C05463=1060.017,236.788,408.491,172.800,33.286,156.181
C05464=1060.024,237.036,408.463,172.802,33.289,156.182
C05465=1060.030,237.285,408.436,172.804,33.293,156.182
C05466=1060.036,237.533,408.408,172.807,33.297,156.183
C05467=1060.042,237.782,408.380,172.809,33.301,156.184
C05468=1060.048,238.030,408.353,172.811,33.305,156.185
C05469=1060.055,238.279,408.326,172.813,33.308,156.185
C05470=1060.061,238.527,408.298,172.815,33.312,156.186
C05471=1060.067,238.775,408.270,172.818,33.316,156.187
C05472=1060.073,239.024,408.243,172.820,33.320,156.188
C05473=1060.079,239.273,408.215,172.822,33.324,156.188
C05474=1060.085,239.521,408.187,172.824,33.328,156.189
C05475=1060.092,239.769,408.160,172.827,33.331,156.190
C05476=1060.098,240.017,408.132,172.829,33.335,156.190
C05477=1060.104,240.266,408.105,172.831,33.339,156.191
C05478=1060.110,240.515,408.077,172.833,33.343,156.192
C05479=1060.116,240.762,408.050,172.836,33.347,156.193
C05480=1060.122,241.011,408.021,172.838,33.350,156.193
C05481=1060.129,241.260,407.994,172.840,33.354,156.194
C05482=1060.135,241.507,407.966,172.842,33.358,156.195
C05483=1060.141,241.757,407.939,172.846,33.362,156.195
C05484=1060.147,242.005,407.911,172.848,33.365,156.196
C05485=1060.154,242.254,407.883,172.850,33.370,156.197
C05486=1060.159,242.502,407.855,172.852,33.373,156.198
C05487=1060.165,242.750,407.827,172.855,33.377,156.198
C05488=1060.171,242.998,407.800,172.857,33.381,156.199
C05489=1060.177,243.247,407.771,172.859,33.385,156.200
C05490=1060.184,243.495,407.743,172.861,33.389,156.201
C05491=1060.189,243.743,407.716,172.864,33.393,156.201
C05492=1060.196,243.992,407.688,172.866,33.396,156.202
C05493=1060.202,244.241,407.659,172.868,33.400,156.203
C05494=1060.209,244.489,407.632,172.870,33.404,156.204
C05495=1060.214,244.737,407.604,172.873,33.408,156.204
C05496=1060.221,244.986,407.576,172.875,33.412,156.205
C05497=1060.227,245.234,407.548,172.877,33.416,156.206
C05498=1060.232,245.482,407.520,172.880,33.420,156.206
C05499=1060.239,245.730,407.491,172.882,33.423,156.207
C05500=1060.245,245.979,407.463,172.885,33.427,156.208
C05501=1060.252,246.227,407.435,172.887,33.431,156.209
C05502=1060.257,246.475,407.407,172.890,33.435,156.209
C05503=1060.263,246.724,407.379,172.892,33.438,156.210
C05504=1060.270,246.973,407.351,172.894,33.443,156.211
C05505=1060.276,247.221,407.322,172.897,33.446,156.212
C05506=1060.281,247.469,407.294,172.899,33.451,156.212
C05507=1060.287,247.718,407.266,172.901,33.454,156.213
C05508=1060.293,247.966,407.238,172.904,33.458,156.214
C05509=1060.300,248.213,407.210,172.906,33.462,156.215
C05510=1060.305,248.462,407.181,172.908,33.466,156.215
C05511=1060.311,248.690,407.156,172.910,33.469,156.216
C05512=1060.316,248.917,407.130,172.912,33.473,156.217
C05513=1060.322,249.144,407.103,172.914,33.477,156.217
C05514=1060.327,249.372,407.078,172.917,33.480,156.218
C05515=1060.333,249.599,407.051,172.920,33.483,156.219
C05516=1060.338,249.825,407.025,172.922,33.487,156.219
C05517=1060.344,250.053,406.999,172.924,33.491,156.220
C05518=1060.350,250.281,406.974,172.926,33.494,156.221
C05519=1060.355,250.528,406.945,172.928,33.498,156.221
C05520=1060.361,250.777,406.917,172.931,33.502,156.222
C05521=1060.368,251.025,406.889,172.933,33.506,156.223
C05522=1060.374,251.273,406.860,172.935,33.509,156.224
C05523=1060.380,251.522,406.832,172.938,33.513,156.224
C05524=1060.386,251.770,406.803,172.940,33.517,156.225
C05525=1060.392,252.018,406.775,172.942,33.521,156.226
C05526=1060.398,252.267,406.745,172.945,33.525,156.227
C05527=1060.405,252.515,406.718,172.947,33.529,156.227
C05528=1060.411,252.763,406.689,172.950,33.532,156.228
C05529=1060.417,253.012,406.660,172.953,33.536,156.229
C05530=1060.423,253.260,406.631,172.955,33.540,156.230
C05531=1060.428,253.508,406.603,172.958,33.544,156.230
C05532=1060.435,253.756,406.574,172.960,33.548,156.231
C05533=1060.441,254.005,406.546,172.962,33.552,156.232
C05534=1060.448,254.253,406.518,172.965,33.555,156.232
C05535=1060.454,254.502,406.489,172.967,33.559,156.233
C05536=1060.460,254.750,406.460,172.970,33.563,156.234
C05537=1060.466,254.998,406.432,172.972,33.567,156.235
C05538=1060.472,255.247,406.403,172.974,33.571,156.235
C05539=1060.478,255.495,406.374,172.977,33.574,156.236
C05540=1060.484,255.743,406.345,172.979,33.578,156.237
C05541=1060.490,255.992,406.316,172.983,33.582,156.238
C05542=1060.497,256.239,406.288,172.985,33.586,156.238
C05543=1060.503,256.488,406.260,172.987,33.589,156.239
C05544=1060.510,256.736,406.231,172.990,33.594,156.240
C05545=1060.516,256.984,406.202,172.992,33.597,156.240
C05546=1060.522,257.233,406.173,172.995,33.601,156.241
C05547=1060.528,257.481,406.144,172.997,33.605,156.242
C05548=1060.534,257.729,406.115,172.999,33.609,156.243
C05549=1060.541,257.978,406.086,173.002,33.612,156.243
C05550=1060.547,258.226,406.058,173.004,33.616,156.244
C05551=1060.553,258.474,406.029,173.007,33.620,156.245
C05552=1060.560,258.722,406.000,173.009,33.624,156.246
C05553=1060.566,258.970,405.971,173.013,33.628,156.246
C05554=1060.572,259.218,405.942,173.015,33.631,156.247
C05555=1060.578,259.467,405.914,173.017,33.635,156.248
C05556=1060.584,259.715,405.885,173.020,33.639,156.249
C05557=1060.591,259.964,405.856,173.022,33.643,156.249
C05558=1060.597,260.212,405.827,173.025,33.646,156.250
C05559=1060.603,260.460,405.798,173.027,33.650,156.251
C05560=1060.609,260.708,405.769,173.030,33.654,156.251
C05561=1060.616,260.956,405.740,173.032,33.658,156.252
C05562=1060.622,261.204,405.711,173.035,33.662,156.253
C05563=1060.628,261.453,405.682,173.037,33.665,156.254
C05564=1060.635,261.702,405.653,173.041,33.669,156.254
C05565=1060.641,261.950,405.624,173.043,33.673,156.255
C05566=1060.647,262.198,405.595,173.045,33.677,156.256
C05567=1060.653,262.424,405.568,173.048,33.680,156.256
C05568=1060.659,262.650,405.542,173.050,33.683,156.257
C05569=1060.665,262.876,405.516,173.052,33.687,156.258
C05570=1060.671,263.103,405.489,173.055,33.690,156.258
C05571=1060.677,263.329,405.463,173.057,33.694,156.259
C05572=1060.682,263.555,405.436,173.059,33.697,156.260
C05573=1060.687,263.781,405.409,173.061,33.701,156.260
C05574=1060.693,264.007,405.382,173.064,33.704,156.261
C05575=1060.699,264.255,405.353,173.067,33.708,156.262
C05576=1060.705,264.503,405.324,173.069,33.712,156.263
C05577=1060.711,264.752,405.294,173.072,33.716,156.263
C05578=1060.717,264.999,405.265,173.074,33.720,156.264
C05579=1060.724,265.248,405.235,173.077,33.723,156.265
C05580=1060.731,265.496,405.206,173.079,33.727,156.266
C05581=1060.736,265.745,405.177,173.082,33.731,156.266
C05582=1060.742,265.993,405.148,173.084,33.735,156.267
C05583=1060.749,266.240,405.118,173.087,33.739,156.268
C05584=1060.754,266.489,405.088,173.089,33.743,156.268
C05585=1060.761,266.737,405.059,173.093,33.746,156.269
C05586=1060.767,266.986,405.030,173.095,33.750,156.270
C05587=1060.773,267.234,404.999,173.098,33.754,156.271
C05588=1060.780,267.482,404.970,173.100,33.758,156.271
C05589=1060.786,267.730,404.941,173.103,33.762,156.272
C05590=1060.792,267.978,404.911,173.106,33.766,156.273
C05591=1060.798,268.226,404.882,173.108,33.769,156.274
C05592=1060.805,268.475,404.852,173.111,33.773,156.274
C05593=1060.811,268.723,404.822,173.113,33.777,156.275
C05594=1060.817,268.971,404.793,173.117,33.781,156.276
C05595=1060.823,269.219,404.764,173.119,33.785,156.277
C05596=1060.829,269.467,404.734,173.122,33.788,156.277
C05597=1060.836,269.715,404.704,173.124,33.793,156.278
C05598=1060.842,269.963,404.674,173.127,33.796,156.279
C05599=1060.848,270.211,404.645,173.129,33.800,156.280
C05600=1060.854,270.459,404.615,173.132,33.804,156.280
C05601=1060.860,270.708,404.585,173.134,33.808,156.281
C05602=1060.866,270.956,404.555,173.137,33.811,156.282
C05603=1060.872,271.204,404.526,173.140,33.816,156.283
C05604=1060.878,271.452,404.495,173.143,33.819,156.283
C05605=1060.885,271.701,404.466,173.146,33.823,156.284
C05606=1060.891,271.948,404.436,173.148,33.827,156.285
C05607=1060.897,272.197,404.407,173.151,33.831,156.286
C05608=1060.903,272.444,404.376,173.153,33.835,156.286
C05609=1060.910,272.693,404.347,173.156,33.838,156.287
C05610=1060.916,272.941,404.316,173.158,33.843,156.288
C05611=1060.922,273.189,404.287,173.162,33.846,156.289
C05612=1060.928,273.438,404.257,173.165,33.850,156.289
C05613=1060.934,273.686,404.226,173.167,33.854,156.290
C05614=1060.941,273.933,404.197,173.170,33.858,156.291
C05615=1060.946,274.182,404.167,173.172,33.862,156.292
C05616=1060.953,274.430,404.137,173.175,33.866,156.292
C05617=1060.959,274.678,404.107,173.177,33.870,156.293
C05618=1060.965,274.925,404.076,173.180,33.873,156.294
C05619=1060.972,275.174,404.047,173.184,33.878,156.295
C05620=1060.978,275.422,404.016,173.186,33.881,156.295
C05621=1060.984,275.670,403.986,173.189,33.885,156.296
C05622=1060.991,275.918,403.956,173.191,33.889,156.297
C05623=1060.998,276.244,403.916,173.195,33.894,156.298
C05624=1061.006,276.568,403.877,173.198,33.899,156.299
C05625=1061.014,276.894,403.837,173.202,33.904,156.300
C05626=1061.023,277.219,403.798,173.206,33.909,156.301
C05627=1061.029,277.466,403.767,173.209,33.913,156.302
C05628=1061.035,277.715,403.737,173.211,33.917,156.303
C05629=1061.042,277.963,403.707,173.214,33.921,156.303
C05630=1061.047,278.210,403.677,173.217,33.925,156.304
C05631=1061.054,278.459,403.646,173.219,33.929,156.305
C05632=1061.059,278.707,403.616,173.222,33.932,156.305
C05633=1061.067,278.956,403.586,173.226,33.937,156.306
C05634=1061.072,279.203,403.556,173.228,33.940,156.307
C05635=1061.078,279.451,403.525,173.231,33.944,156.308
C05636=1061.085,279.700,403.495,173.233,33.948,156.309
C05637=1061.091,279.947,403.465,173.236,33.952,156.309
C05638=1061.098,280.196,403.434,173.239,33.956,156.310
C05639=1061.104,280.443,403.403,173.241,33.960,156.311
C05640=1061.110,280.691,403.372,173.244,33.964,156.312
C05641=1061.116,280.939,403.342,173.248,33.968,156.312
C05642=1061.122,281.188,403.311,173.250,33.972,156.313
C05643=1061.128,281.436,403.281,173.253,33.976,156.314
C05644=1061.134,281.683,403.251,173.256,33.980,156.315
C05645=1061.140,281.932,403.220,173.258,33.983,156.315
C05646=1061.146,282.180,403.190,173.261,33.987,156.316
C05647=1061.156,282.559,403.143,173.266,33.993,156.317
C05648=1061.166,282.938,403.095,173.270,33.999,156.319
C05649=1061.175,283.317,403.049,173.274,34.005,156.320
C05650=1061.185,283.696,403.002,173.278,34.011,156.321
C05651=1061.191,283.944,402.971,173.281,34.015,156.322
C05652=1061.197,284.192,402.940,173.285,34.019,156.323
C05653=1061.203,284.439,402.909,173.287,34.023,156.323
C05654=1061.210,284.688,402.879,173.290,34.027,156.324
C05655=1061.216,284.936,402.848,173.293,34.031,156.325
C05656=1061.222,285.184,402.817,173.296,34.035,156.326
C05657=1061.228,285.432,402.786,173.298,34.039,156.326
C05658=1061.235,285.679,402.755,173.301,34.043,156.327
C05659=1061.241,285.928,402.724,173.305,34.047,156.328
C05660=1061.247,286.176,402.694,173.307,34.051,156.329
C05661=1061.254,286.424,402.663,173.310,34.055,156.330
C05662=1061.260,286.672,402.632,173.313,34.059,156.330
C05663=1061.266,286.919,402.601,173.316,34.062,156.331
C05664=1061.273,287.168,402.570,173.318,34.067,156.332
C05665=1061.279,287.415,402.539,173.322,34.070,156.333
C05666=1061.285,287.664,402.508,173.325,34.074,156.333
C05667=1061.291,287.912,402.476,173.327,34.078,156.334
C05668=1061.297,288.160,402.446,173.330,34.082,156.335
C05669=1061.304,288.407,402.415,173.333,34.086,156.336
C05670=1061.310,288.656,402.384,173.336,34.090,156.337
C05671=1061.316,288.903,402.353,173.338,34.094,156.337
C05672=1061.323,289.152,402.322,173.342,34.098,156.338
C05673=1061.329,289.399,402.291,173.345,34.102,156.339
C05674=1061.335,289.647,402.259,173.348,34.106,156.340
C05675=1061.340,289.881,402.230,173.350,34.110,156.340
C05676=1061.347,290.114,402.201,173.353,34.114,156.341
C05677=1061.352,290.347,402.171,173.356,34.117,156.342
C05678=1061.358,290.581,402.142,173.359,34.121,156.343
C05679=1061.364,290.815,402.113,173.362,34.125,156.343
C05680=1061.370,291.048,402.083,173.364,34.129,156.344
C05681=1061.376,291.281,402.054,173.367,34.132,156.345
C05682=1061.382,291.515,402.023,173.370,34.136,156.346
C05683=1061.388,291.763,401.993,173.372,34.140,156.347
C05684=1061.394,292.011,401.962,173.376,34.144,156.347
C05685=1061.401,292.259,401.930,173.379,34.148,156.348
C05686=1061.407,292.507,401.898,173.382,34.152,156.349
C05687=1061.413,292.754,401.867,173.384,34.156,156.350
C05688=1061.420,293.002,401.836,173.387,34.160,156.351
C05689=1061.426,293.251,401.804,173.390,34.164,156.351
C05690=1061.432,293.498,401.773,173.394,34.168,156.352
C05691=1061.438,293.746,401.742,173.397,34.172,156.353
C05692=1061.444,293.994,401.710,173.399,34.176,156.354
C05693=1061.451,294.242,401.678,173.402,34.180,156.354
C05694=1061.457,294.489,401.647,173.405,34.184,156.355
C05695=1061.463,294.737,401.615,173.409,34.188,156.356
C05696=1061.470,294.985,401.584,173.412,34.192,156.357
C05697=1061.476,295.233,401.552,173.415,34.196,156.358
C05698=1061.483,295.481,401.520,173.417,34.200,156.359
C05699=1061.488,295.729,401.489,173.420,34.204,156.359
C05700=1061.495,295.977,401.457,173.423,34.209,156.360
C05701=1061.502,296.225,401.426,173.427,34.212,156.361
C05702=1061.508,296.473,401.394,173.430,34.216,156.362
C05703=1061.514,296.721,401.362,173.433,34.221,156.363
C05704=1061.520,296.968,401.331,173.435,34.225,156.363
C05705=1061.526,297.216,401.299,173.438,34.229,156.364
C05706=1061.532,297.464,401.267,173.442,34.233,156.365
C05707=1061.539,297.712,401.235,173.445,34.237,156.366
C05708=1061.544,297.959,401.203,173.448,34.241,156.367
C05709=1061.551,298.207,401.172,173.451,34.245,156.368
C05710=1061.557,298.456,401.139,173.453,34.250,156.368
C05711=1061.563,298.704,401.107,173.457,34.254,156.369
C05712=1061.568,298.951,401.075,173.460,34.258,156.370
C05713=1061.575,299.199,401.044,173.463,34.262,156.371
C05714=1061.581,299.447,401.012,173.466,34.266,156.372
C05715=1061.587,299.694,400.979,173.469,34.270,156.373
C05716=1061.593,299.943,400.947,173.471,34.274,156.373
C05717=1061.600,300.191,400.915,173.475,34.278,156.374
C05718=1061.606,300.437,400.883,173.478,34.282,156.375
C05719=1061.612,300.686,400.851,173.481,34.286,156.376
C05720=1061.618,300.934,400.819,173.484,34.291,156.377
C05721=1061.624,301.181,400.786,173.487,34.295,156.378
C05722=1061.631,301.429,400.755,173.491,34.299,156.378
C05723=1061.637,301.678,400.723,173.494,34.303,156.379
C05724=1061.643,301.925,400.690,173.497,34.307,156.380
C05725=1061.649,302.173,400.658,173.499,34.311,156.381
C05726=1061.656,302.420,400.626,173.503,34.315,156.382
C05727=1061.661,302.668,400.594,173.506,34.320,156.383
C05728=1061.668,302.916,400.561,173.509,34.324,156.383
C05729=1061.674,303.164,400.529,173.512,34.328,156.384
C05730=1061.680,303.412,400.497,173.515,34.332,156.385
C05731=1061.686,303.653,400.465,173.519,34.336,156.386
C05732=1061.693,303.894,400.434,173.522,34.340,156.387
C05733=1061.699,304.134,400.403,173.524,34.344,156.388
C05734=1061.704,304.376,400.371,173.527,34.349,156.388
C05735=1061.711,304.617,400.340,173.530,34.353,156.389
C05736=1061.718,304.858,400.308,173.534,34.357,156.390
C05737=1061.723,305.099,400.276,173.537,34.360,156.391
C05738=1061.729,305.340,400.245,173.540,34.365,156.392
C05739=1061.735,305.587,400.213,173.543,34.369,156.393
C05740=1061.741,305.836,400.181,173.546,34.373,156.393
C05741=1061.748,306.084,400.147,173.550,34.377,156.394
C05742=1061.755,306.331,400.115,173.553,34.381,156.395
C05743=1061.761,306.579,400.083,173.556,34.386,156.396
C05744=1061.768,306.827,400.051,173.559,34.390,156.397
C05745=1061.774,307.075,400.018,173.563,34.394,156.398
C05746=1061.780,307.322,399.985,173.566,34.398,156.399
C05747=1061.786,307.570,399.953,173.568,34.402,156.399
C05748=1061.793,307.818,399.920,173.571,34.407,156.400
C05749=1061.800,308.065,399.888,173.574,34.411,156.401
C05750=1061.806,308.313,399.855,173.578,34.415,156.402
C05751=1061.812,308.560,399.823,173.581,34.419,156.403
C05752=1061.818,308.808,399.790,173.584,34.423,156.404
C05753=1061.825,309.057,399.758,173.587,34.427,156.404
C05754=1061.831,309.305,399.725,173.591,34.431,156.405
C05755=1061.838,309.552,399.692,173.594,34.436,156.406
C05756=1061.844,309.800,399.659,173.597,34.440,156.407
C05757=1061.850,310.047,399.627,173.600,34.444,156.408
C05758=1061.858,310.295,399.594,173.603,34.448,156.409
C05759=1061.864,310.543,399.561,173.608,34.453,156.410
C05760=1061.870,310.790,399.529,173.611,34.457,156.410
C05761=1061.877,311.038,399.496,173.614,34.461,156.411
C05762=1061.883,311.286,399.463,173.617,34.465,156.412
C05763=1061.890,311.534,399.430,173.621,34.469,156.413
C05764=1061.896,311.782,399.397,173.624,34.474,156.414
C05765=1061.902,312.029,399.364,173.627,34.478,156.415
C05766=1061.909,312.277,399.332,173.630,34.482,156.416
C05767=1061.916,312.525,399.299,173.634,34.486,156.416
C05768=1061.922,312.773,399.266,173.637,34.490,156.417
C05769=1061.928,313.020,399.233,173.640,34.495,156.418
C05770=1061.935,313.268,399.199,173.643,34.499,156.419
C05771=1061.942,313.515,399.167,173.647,34.503,156.420
C05772=1061.948,313.763,399.134,173.650,34.507,156.421
C05773=1061.955,314.011,399.101,173.653,34.512,156.422
C05774=1061.961,314.259,399.068,173.656,34.516,156.423
C05775=1061.967,314.506,399.034,173.660,34.520,156.424
C05776=1061.973,314.754,399.001,173.663,34.525,156.424
C05777=1061.979,315.002,398.968,173.666,34.529,156.425
C05778=1061.986,315.249,398.934,173.669,34.534,156.426
C05779=1061.992,315.497,398.901,173.673,34.538,156.427
C05780=1061.998,315.745,398.868,173.676,34.543,156.428
C05781=1062.005,315.992,398.834,173.679,34.547,156.429
C05782=1062.011,316.240,398.801,173.683,34.552,156.430
C05783=1062.017,316.487,398.767,173.687,34.556,156.431
C05784=1062.023,316.735,398.734,173.690,34.560,156.432
C05785=1062.029,316.983,398.701,173.693,34.564,156.433
C05786=1062.036,317.231,398.667,173.696,34.569,156.434
C05787=1062.042,317.473,398.635,173.700,34.573,156.434
C05788=1062.048,317.716,398.601,173.703,34.578,156.435
C05789=1062.054,317.960,398.568,173.706,34.582,156.436
C05790=1062.060,318.202,398.535,173.709,34.586,156.437
C05791=1062.067,318.445,398.503,173.713,34.591,156.438
C05792=1062.073,318.688,398.470,173.716,34.595,156.439
C05793=1062.079,318.932,398.436,173.719,34.600,156.440
C05794=1062.085,319.174,398.404,173.722,34.604,156.441
C05795=1062.091,319.423,398.370,173.726,34.608,156.442
C05796=1062.097,319.670,398.336,173.729,34.612,156.443
C05797=1062.105,319.917,398.303,173.732,34.617,156.444
C05798=1062.110,320.165,398.269,173.736,34.621,156.444
C05799=1062.117,320.412,398.236,173.740,34.626,156.445
C05800=1062.123,320.660,398.201,173.743,34.631,156.446
C05801=1062.129,320.908,398.169,173.746,34.635,156.447
C05802=1062.136,321.156,398.134,173.750,34.639,156.448
C05803=1062.143,321.403,398.101,173.753,34.644,156.449
C05804=1062.149,321.651,398.066,173.756,34.648,156.450
C05805=1062.155,321.898,398.034,173.760,34.653,156.451
C05806=1062.162,322.146,397.999,173.764,34.657,156.452
C05807=1062.168,322.393,397.966,173.767,34.662,156.453
C05808=1062.175,322.641,397.931,173.770,34.666,156.454
C05809=1062.181,322.889,397.897,173.774,34.670,156.455
C05810=1062.188,323.137,397.864,173.777,34.675,156.456
C05811=1062.193,323.384,397.830,173.780,34.680,156.457
C05812=1062.201,323.632,397.796,173.785,34.684,156.457
C05813=1062.206,323.879,397.762,173.788,34.688,156.458
C05814=1062.214,324.127,397.728,173.791,34.693,156.459
C05815=1062.220,324.375,397.694,173.794,34.698,156.460
C05816=1062.226,324.622,397.660,173.798,34.702,156.461
C05817=1062.233,324.870,397.626,173.802,34.707,156.462
C05818=1062.239,325.117,397.592,173.805,34.711,156.463
C05819=1062.246,325.365,397.558,173.809,34.716,156.464
C05820=1062.253,325.613,397.524,173.812,34.720,156.465
C05821=1062.259,325.860,397.490,173.815,34.725,156.466
C05822=1062.266,326.108,397.456,173.820,34.729,156.467
C05823=1062.272,326.356,397.421,173.823,34.734,156.468
C05824=1062.279,326.603,397.388,173.826,34.738,156.469
C05825=1062.285,326.851,397.354,173.829,34.743,156.470
C05826=1062.292,327.099,397.319,173.833,34.747,156.471
C05827=1062.298,327.346,397.286,173.837,34.752,156.472
C05828=1062.305,327.593,397.251,173.840,34.756,156.473
C05829=1062.312,327.841,397.216,173.844,34.761,156.474
C05830=1062.318,328.088,397.183,173.847,34.765,156.475
C05831=1062.325,328.336,397.148,173.851,34.770,156.475
C05832=1062.331,328.584,397.114,173.855,34.775,156.476
C05833=1062.339,328.831,397.079,173.858,34.779,156.477
C05834=1062.344,329.078,397.045,173.861,34.783,156.478
C05835=1062.351,329.326,397.011,173.866,34.788,156.479
C05836=1062.358,329.574,396.977,173.869,34.793,156.480
C05837=1062.365,329.821,396.942,173.872,34.797,156.481
C05838=1062.371,330.069,396.907,173.876,34.802,156.482
C05839=1062.378,330.316,396.874,173.880,34.807,156.483
C05840=1062.385,330.564,396.839,173.883,34.811,156.484
C05841=1062.391,330.812,396.804,173.886,34.816,156.485
C05842=1062.398,331.060,396.770,173.891,34.821,156.486
C05843=1062.404,331.299,396.736,173.894,34.825,156.487
C05844=1062.411,331.540,396.703,173.897,34.830,156.488
C05845=1062.417,331.780,396.669,173.901,34.835,156.489
C05846=1062.423,332.020,396.635,173.904,34.839,156.490
C05847=1062.429,332.260,396.602,173.908,34.843,156.491
C05848=1062.436,332.500,396.568,173.912,34.848,156.492
C05849=1062.442,332.740,396.534,173.915,34.853,156.493
C05850=1062.448,332.980,396.501,173.918,34.857,156.494
C05851=1062.454,333.228,396.465,173.923,34.862,156.495
C05852=1062.461,333.474,396.430,173.926,34.867,156.496
C05853=1062.467,333.722,396.396,173.929,34.872,156.497
C05854=1062.474,333.970,396.361,173.934,34.876,156.498
C05855=1062.481,334.217,396.326,173.937,34.881,156.499
C05856=1062.487,334.465,396.291,173.940,34.886,156.500
C05857=1062.494,334.713,396.256,173.944,34.891,156.501
C05858=1062.501,334.960,396.221,173.948,34.895,156.502
C05859=1062.507,335.208,396.187,173.952,34.900,156.503
C05860=1062.513,335.455,396.152,173.956,34.905,156.504
C05861=1062.520,335.702,396.117,173.959,34.910,156.505
C05862=1062.527,335.949,396.082,173.963,34.914,156.506
C05863=1062.534,336.197,396.046,173.967,34.919,156.507
C05864=1062.540,336.445,396.012,173.970,34.924,156.508
C05865=1062.547,336.692,395.977,173.974,34.929,156.509
C05866=1062.553,336.940,395.941,173.978,34.934,156.510
C05867=1062.560,337.187,395.906,173.981,34.939,156.511
C05868=1062.566,337.434,395.871,173.985,34.943,156.512
C05869=1062.573,337.682,395.836,173.989,34.948,156.513
C05870=1062.579,337.929,395.800,173.992,34.953,156.514
C05871=1062.586,338.177,395.765,173.997,34.958,156.515
C05872=1062.593,338.424,395.730,174.000,34.963,156.516
C05873=1062.599,338.672,395.694,174.004,34.968,156.518
C05874=1062.605,338.919,395.659,174.008,34.973,156.519
C05875=1062.612,339.167,395.624,174.011,34.978,156.520
C05876=1062.618,339.414,395.588,174.016,34.983,156.521
C05877=1062.625,339.662,395.553,174.019,34.988,156.522
C05878=1062.632,339.909,395.518,174.023,34.993,156.523
C05879=1062.639,340.156,395.483,174.027,34.997,156.524
C05880=1062.645,340.403,395.446,174.030,35.003,156.525
C05881=1062.652,340.651,395.411,174.035,35.007,156.526
C05882=1062.658,340.898,395.376,174.038,35.012,156.527
C05883=1062.664,341.146,395.340,174.041,35.018,156.528
C05884=1062.671,341.393,395.305,174.046,35.022,156.529
C05885=1062.678,341.640,395.269,174.049,35.027,156.530
C05886=1062.684,341.888,395.233,174.054,35.033,156.531
C05887=1062.691,342.135,395.198,174.057,35.037,156.532
C05888=1062.698,342.383,395.162,174.061,35.042,156.534
C05889=1062.705,342.630,395.126,174.065,35.047,156.535
C05890=1062.712,342.877,395.091,174.069,35.052,156.536
C05891=1062.718,343.125,395.055,174.073,35.057,156.537
C05892=1062.725,343.372,395.020,174.077,35.062,156.538
C05893=1062.731,343.620,394.984,174.080,35.068,156.539
C05894=1062.738,343.867,394.948,174.085,35.072,156.540
C05895=1062.744,344.115,394.912,174.088,35.077,156.541
C05896=1062.751,344.361,394.876,174.092,35.083,156.542
C05897=1062.758,344.609,394.840,174.096,35.088,156.543
C05898=1062.765,344.856,394.805,174.100,35.093,156.545
C05899=1062.771,345.094,394.770,174.104,35.098,156.546
C05900=1062.778,345.332,394.735,174.107,35.103,156.547
C05901=1062.783,345.569,394.701,174.112,35.108,156.548
C05902=1062.790,345.807,394.666,174.115,35.112,156.549
C05903=1062.796,346.045,394.632,174.119,35.117,156.550
C05904=1062.802,346.282,394.597,174.123,35.123,156.551
C05905=1062.809,346.520,394.562,174.126,35.127,156.552
C05906=1062.815,346.758,394.528,174.130,35.132,156.553
C05907=1062.822,347.005,394.491,174.134,35.138,156.554
C05908=1062.829,347.252,394.455,174.138,35.143,156.555
C05909=1062.835,347.500,394.419,174.142,35.148,156.556
C05910=1062.842,347.748,394.383,174.147,35.153,156.558
C05911=1062.849,347.994,394.347,174.150,35.158,156.559
C05912=1062.855,348.241,394.310,174.154,35.163,156.560
C05913=1062.862,348.490,394.274,174.158,35.169,156.561
C05914=1062.869,348.736,394.239,174.162,35.174,156.562
C05915=1062.875,348.983,394.202,174.166,35.179,156.563
C05916=1062.882,349.231,394.165,174.170,35.184,156.564
C05917=1062.888,349.478,394.129,174.174,35.190,156.566
C05918=1062.895,349.725,394.093,174.178,35.195,156.567
C05919=1062.902,349.973,394.056,174.183,35.200,156.568
C05920=1062.909,350.220,394.020,174.186,35.205,156.569
C05921=1062.916,350.467,393.984,174.191,35.211,156.570
C05922=1062.923,350.714,393.947,174.194,35.216,156.571
C05923=1062.929,350.961,393.911,174.198,35.221,156.573
C05924=1062.936,351.209,393.874,174.203,35.227,156.574
C05925=1062.943,351.456,393.838,174.206,35.232,156.575
C05926=1062.950,351.704,393.801,174.211,35.237,156.576
C05927=1062.956,351.951,393.765,174.214,35.243,156.577
C05928=1062.963,352.198,393.728,174.219,35.248,156.578
C05929=1062.970,352.446,393.691,174.223,35.253,156.580
C05930=1062.976,352.693,393.655,174.227,35.258,156.581
C05931=1062.983,352.940,393.617,174.231,35.264,156.582
C05932=1062.990,353.187,393.581,174.235,35.269,156.583
C05933=1062.996,353.434,393.545,174.239,35.275,156.584
C05934=1063.003,353.682,393.508,174.244,35.280,156.586
C05935=1063.009,353.928,393.471,174.247,35.286,156.587
C05936=1063.016,354.176,393.434,174.252,35.291,156.588
C05937=1063.023,354.423,393.397,174.256,35.297,156.589
C05938=1063.030,354.670,393.360,174.260,35.302,156.590
C05939=1063.036,354.917,393.323,174.264,35.307,156.592
C05940=1063.043,355.165,393.287,174.269,35.313,156.593
C05941=1063.050,355.411,393.249,174.272,35.319,156.594
C05942=1063.057,355.659,393.213,174.277,35.324,156.595
C05943=1063.063,355.905,393.175,174.281,35.330,156.596
C05944=1063.070,356.153,393.139,174.285,35.335,156.598
C05945=1063.078,356.400,393.101,174.289,35.340,156.599
C05946=1063.084,356.647,393.065,174.294,35.346,156.600
C05947=1063.091,356.894,393.027,174.297,35.352,156.601
C05948=1063.098,357.142,392.991,174.302,35.357,156.603
C05949=1063.105,357.389,392.953,174.306,35.363,156.604
C05950=1063.112,357.636,392.916,174.311,35.368,156.605
C05951=1063.118,357.883,392.879,174.314,35.374,156.606
C05952=1063.126,358.130,392.842,174.319,35.379,156.608
C05953=1063.133,358.378,392.805,174.323,35.385,156.609
C05954=1063.139,358.624,392.768,174.327,35.391,156.610
C05955=1063.146,358.864,392.731,174.331,35.396,156.611
C05956=1063.152,359.104,392.695,174.336,35.401,156.612
C05957=1063.159,359.343,392.659,174.340,35.407,156.614
C05958=1063.166,359.584,392.622,174.344,35.413,156.615
C05959=1063.173,359.823,392.586,174.349,35.418,156.616
C05960=1063.179,360.063,392.550,174.352,35.423,156.617
C05961=1063.186,360.303,392.513,174.357,35.429,156.619
C05962=1063.193,360.543,392.478,174.361,35.435,156.620
C05963=1063.199,360.790,392.439,174.365,35.440,156.621
C05964=1063.206,361.037,392.402,174.369,35.446,156.622
C05965=1063.213,361.284,392.365,174.374,35.452,156.624
C05966=1063.220,361.531,392.327,174.378,35.457,156.625
C05967=1063.227,361.778,392.289,174.382,35.463,156.626
C05968=1063.233,362.025,392.252,174.387,35.469,156.628
C05969=1063.241,362.272,392.214,174.391,35.475,156.629
C05970=1063.247,362.520,392.176,174.396,35.480,156.630
C05971=1063.254,362.767,392.139,174.400,35.486,156.631
C05972=1063.261,363.013,392.102,174.404,35.492,156.633
C05973=1063.268,363.260,392.064,174.408,35.498,156.634
C05974=1063.275,363.508,392.026,174.413,35.504,156.635
C05975=1063.282,363.754,391.988,174.418,35.509,156.637
C05976=1063.290,364.001,391.950,174.422,35.515,156.638
C05977=1063.296,364.249,391.912,174.426,35.521,156.639
C05978=1063.303,364.495,391.875,174.430,35.527,156.641
C05979=1063.309,364.743,391.837,174.435,35.533,156.642
C05980=1063.317,364.989,391.798,174.440,35.539,156.643
C05981=1063.323,365.237,391.760,174.444,35.545,156.645
C05982=1063.330,365.484,391.722,174.449,35.551,156.646
C05983=1063.337,365.731,391.684,174.452,35.557,156.647
C05984=1063.343,365.977,391.646,174.457,35.563,156.649
C05985=1063.351,366.224,391.608,174.462,35.569,156.650
C05986=1063.357,366.471,391.570,174.466,35.575,156.652
C05987=1063.365,366.718,391.532,174.471,35.581,156.653
C05988=1063.371,366.965,391.494,174.475,35.587,156.654
C05989=1063.378,367.212,391.455,174.480,35.593,156.656
C05990=1063.385,367.459,391.417,174.485,35.599,156.657
C05991=1063.392,367.706,391.378,174.488,35.605,156.658
C05992=1063.399,367.953,391.341,174.493,35.611,156.660
C05993=1063.406,368.200,391.302,174.498,35.617,156.661
C05994=1063.413,368.447,391.264,174.502,35.623,156.662
C05995=1063.420,368.694,391.226,174.507,35.629,156.664
C05996=1063.427,368.941,391.187,174.512,35.635,156.665
C05997=1063.434,369.188,391.149,174.516,35.641,156.667
C05998=1063.441,369.435,391.110,174.521,35.647,156.668
C05999=1063.448,369.682,391.072,174.526,35.653,156.669
C06000=1063.455,369.928,391.033,174.530,35.660,156.671
C06001=1063.462,370.175,390.995,174.535,35.666,156.672
C06002=1063.470,370.422,390.957,174.539,35.672,156.674
C06003=1063.476,370.669,390.918,174.544,35.678,156.675
C06004=1063.483,370.916,390.879,174.549,35.684,156.676
C06005=1063.491,371.162,390.841,174.553,35.690,156.678
C06006=1063.497,371.410,390.803,174.558,35.696,156.679
C06007=1063.504,371.656,390.764,174.562,35.703,156.681
C06008=1063.512,371.903,390.726,174.567,35.709,156.682
C06009=1063.519,372.150,390.687,174.571,35.715,156.684
C06010=1063.526,372.397,390.648,174.576,35.722,156.685
C06011=1063.533,372.648,390.609,174.582,35.728,156.686
C06012=1063.541,372.898,390.569,174.586,35.734,156.688
C06013=1063.548,373.148,390.530,174.591,35.741,156.689
C06014=1063.554,373.399,390.490,174.596,35.747,156.691
C06015=1063.561,373.646,390.451,174.600,35.754,156.692
C06016=1063.568,373.893,390.412,174.605,35.760,156.694
C06017=1063.575,374.139,390.373,174.610,35.767,156.695
C06018=1063.582,374.386,390.334,174.615,35.773,156.697
C06019=1063.589,374.633,390.295,174.619,35.779,156.698
C06020=1063.597,374.880,390.257,174.624,35.786,156.700
C06021=1063.604,375.126,390.217,174.629,35.792,156.701
C06022=1063.611,375.373,390.178,174.633,35.798,156.703
C06023=1063.618,375.620,390.139,174.638,35.805,156.704
C06024=1063.625,375.867,390.099,174.643,35.812,156.706
C06025=1063.632,376.113,390.061,174.648,35.818,156.707
C06026=1063.639,376.360,390.022,174.652,35.825,156.709
C06027=1063.646,376.606,389.982,174.657,35.831,156.710
C06028=1063.654,376.854,389.943,174.662,35.838,156.712
C06029=1063.661,377.100,389.903,174.667,35.844,156.713
C06030=1063.667,377.347,389.865,174.671,35.851,156.715
C06031=1063.675,377.594,389.825,174.677,35.857,156.716
C06032=1063.682,377.841,389.786,174.682,35.864,156.718
C06033=1063.689,378.087,389.746,174.687,35.871,156.719
C06034=1063.697,378.334,389.707,174.692,35.877,156.721
C06035=1063.704,378.581,389.668,174.696,35.884,156.723
C06036=1063.711,378.828,389.628,174.701,35.890,156.724
C06037=1063.718,379.074,389.589,174.706,35.897,156.725
C06038=1063.725,379.321,389.549,174.711,35.903,156.727
C06039=1063.733,379.567,389.509,174.716,35.910,156.729
C06040=1063.740,379.814,389.470,174.721,35.917,156.730
C06041=1063.747,380.062,389.430,174.726,35.924,156.732
C06042=1063.754,380.308,389.390,174.731,35.930,156.733
C06043=1063.762,380.555,389.350,174.736,35.937,156.735
C06044=1063.769,380.801,389.311,174.740,35.944,156.736
C06045=1063.776,381.048,389.271,174.746,35.950,156.738
C06046=1063.784,381.294,389.231,174.751,35.957,156.740
C06047=1063.790,381.542,389.192,174.756,35.964,156.741
C06048=1063.797,381.788,389.152,174.761,35.971,156.743
C06049=1063.805,382.034,389.112,174.766,35.978,156.745
C06050=1063.812,382.281,389.071,174.770,35.984,156.746
C06051=1063.819,382.527,389.032,174.776,35.992,156.748
C06052=1063.827,382.774,388.992,174.781,35.998,156.749
C06053=1063.833,383.020,388.952,174.786,36.005,156.751
C06054=1063.841,383.267,388.912,174.791,36.013,156.753
C06055=1063.848,383.514,388.872,174.797,36.019,156.754
C06056=1063.855,383.761,388.832,174.802,36.026,156.756
C06057=1063.863,384.007,388.791,174.806,36.034,156.758
C06058=1063.870,384.253,388.752,174.811,36.040,156.759
C06059=1063.877,384.500,388.711,174.817,36.047,156.761
C06060=1063.884,384.747,388.671,174.822,36.054,156.763
C06061=1063.891,384.993,388.630,174.827,36.062,156.764
C06062=1063.899,385.240,388.590,174.832,36.068,156.766
C06063=1063.906,385.486,388.551,174.838,36.075,156.767
C06064=1063.914,385.733,388.510,174.843,36.083,156.769
C06065=1063.921,385.980,388.470,174.847,36.090,156.771
C06066=1063.928,386.226,388.429,174.852,36.097,156.773
C06067=1063.936,386.507,388.383,174.858,36.105,156.775
C06068=1063.945,386.788,388.337,174.864,36.113,156.776
C06069=1063.953,387.070,388.290,174.870,36.122,156.778
C06070=1063.962,387.351,388.244,174.877,36.130,156.780
C06071=1063.969,387.597,388.204,174.882,36.137,156.782
C06072=1063.976,387.844,388.164,174.887,36.144,156.784
C06073=1063.984,388.090,388.123,174.892,36.151,156.785
C06074=1063.992,388.337,388.082,174.898,36.158,156.787
C06075=1063.999,388.584,388.042,174.903,36.165,156.789
C06076=1064.007,388.829,388.002,174.908,36.173,156.791
C06077=1064.014,389.076,387.960,174.914,36.180,156.792
C06078=1064.022,389.322,387.920,174.919,36.187,156.794
C06079=1064.029,389.570,387.879,174.925,36.195,156.796
C06080=1064.037,389.816,387.839,174.930,36.202,156.798
C06081=1064.044,390.062,387.797,174.935,36.209,156.799
C06082=1064.052,390.309,387.757,174.941,36.217,156.801
C06083=1064.060,390.555,387.715,174.946,36.224,156.803
C06084=1064.066,390.801,387.675,174.952,36.232,156.805
C06085=1064.074,391.047,387.634,174.957,36.239,156.807
C06086=1064.082,391.294,387.593,174.962,36.246,156.808
C06087=1064.089,391.541,387.552,174.968,36.254,156.810
C06088=1064.097,391.787,387.511,174.973,36.262,156.812
C06089=1064.104,392.034,387.470,174.979,36.269,156.814
C06090=1064.111,392.280,387.428,174.984,36.277,156.816
C06091=1064.119,392.527,387.387,174.990,36.285,156.817
C06092=1064.127,392.773,387.347,174.995,36.292,156.819
C06093=1064.134,393.019,387.305,175.001,36.299,156.821
C06094=1064.142,393.266,387.263,175.006,36.307,156.823
C06095=1064.149,393.512,387.222,175.012,36.315,156.825
C06096=1064.157,393.758,387.182,175.017,36.322,156.827
C06097=1064.165,394.004,387.140,175.023,36.330,156.828
C06098=1064.172,394.251,387.098,175.028,36.338,156.830
C06099=1064.179,394.497,387.056,175.034,36.346,156.832
C06100=1064.187,394.744,387.015,175.039,36.353,156.834
C06101=1064.194,394.990,386.974,175.046,36.361,156.836
C06102=1064.202,395.236,386.932,175.051,36.369,156.838
C06103=1064.209,395.483,386.891,175.057,36.377,156.840
C06104=1064.216,395.729,386.849,175.062,36.385,156.842
C06105=1064.224,395.976,386.807,175.068,36.392,156.843
C06106=1064.232,396.222,386.765,175.073,36.400,156.845
C06107=1064.240,396.468,386.724,175.079,36.408,156.847
C06108=1064.248,396.714,386.683,175.085,36.416,156.849
C06109=1064.255,396.960,386.641,175.090,36.424,156.851
C06110=1064.263,397.207,386.598,175.096,36.432,156.853
C06111=1064.271,397.453,386.557,175.102,36.439,156.855
C06112=1064.278,397.699,386.515,175.108,36.448,156.857
C06113=1064.286,397.945,386.473,175.114,36.456,156.859
C06114=1064.293,398.192,386.430,175.119,36.464,156.861
C06115=1064.301,398.439,386.389,175.125,36.472,156.863
C06116=1064.308,398.685,386.347,175.130,36.480,156.865
C06117=1064.316,398.932,386.305,175.137,36.488,156.867
C06118=1064.324,399.178,386.263,175.143,36.496,156.869
C06119=1064.332,399.424,386.221,175.148,36.504,156.871
C06120=1064.339,399.670,386.179,175.154,36.513,156.873
C06121=1064.347,399.917,386.136,175.160,36.521,156.875
C06122=1064.354,400.163,386.094,175.165,36.529,156.877
C06123=1064.364,400.460,386.043,175.173,36.539,156.879
C06124=1064.373,400.759,385.992,175.180,36.549,156.882
C06125=1064.383,401.056,385.941,175.187,36.558,156.884
C06126=1064.392,401.353,385.889,175.194,36.569,156.887
C06127=1064.400,401.600,385.847,175.201,36.577,156.889
C06128=1064.408,401.846,385.805,175.206,36.585,156.891
C06129=1064.416,402.092,385.763,175.212,36.594,156.893
C06130=1064.423,402.338,385.720,175.218,36.602,156.895
C06131=1064.431,402.585,385.677,175.225,36.610,156.897
C06132=1064.439,402.831,385.635,175.230,36.619,156.899
C06133=1064.446,403.077,385.592,175.236,36.627,156.901
C06134=1064.455,403.324,385.549,175.242,36.636,156.903
C06135=1064.463,403.569,385.507,175.249,36.644,156.905
C06136=1064.470,403.816,385.464,175.255,36.653,156.907
C06137=1064.478,404.062,385.422,175.260,36.661,156.910
C06138=1064.486,404.308,385.379,175.267,36.670,156.912
C06139=1064.494,404.555,385.335,175.273,36.679,156.914
C06140=1064.501,404.801,385.293,175.279,36.687,156.916
C06141=1064.509,405.047,385.250,175.286,36.696,156.918
C06142=1064.518,405.293,385.207,175.291,36.704,156.920
C06143=1064.525,405.539,385.164,175.297,36.713,156.922
C06144=1064.533,405.785,385.121,175.304,36.722,156.925
C06145=1064.541,406.032,385.078,175.310,36.731,156.927
C06146=1064.549,406.277,385.035,175.316,36.739,156.929
C06147=1064.556,406.524,384.992,175.323,36.748,156.931
C06148=1064.564,406.770,384.948,175.329,36.757,156.933
C06149=1064.572,407.016,384.905,175.336,36.766,156.936
C06150=1064.580,407.262,384.862,175.341,36.775,156.938
C06151=1064.587,407.508,384.818,175.347,36.784,156.940
C06152=1064.596,407.755,384.775,175.354,36.793,156.942
C06153=1064.604,408.001,384.732,175.360,36.801,156.944
C06154=1064.612,408.246,384.689,175.367,36.810,156.947
C06155=1064.619,408.493,384.645,175.373,36.820,156.949
C06156=1064.627,408.738,384.601,175.380,36.829,156.951
C06157=1064.635,408.985,384.558,175.386,36.838,156.954
C06158=1064.644,409.231,384.514,175.393,36.847,156.956
C06159=1064.651,409.477,384.471,175.399,36.856,156.958
C06160=1064.659,409.723,384.427,175.406,36.865,156.960
C06161=1064.668,409.969,384.384,175.412,36.874,156.963
C06162=1064.676,410.215,384.340,175.418,36.883,156.965
C06163=1064.684,410.462,384.296,175.425,36.892,156.967
C06164=1064.692,410.707,384.253,175.431,36.901,156.970
C06165=1064.700,410.953,384.209,175.438,36.911,156.972
C06166=1064.708,411.199,384.165,175.445,36.920,156.974
C06167=1064.716,411.446,384.121,175.452,36.929,156.977
C06168=1064.725,411.691,384.077,175.459,36.938,156.979
C06169=1064.733,411.937,384.034,175.465,36.948,156.981
C06170=1064.741,412.183,383.989,175.472,36.957,156.984
C06171=1064.748,412.429,383.946,175.478,36.966,156.986
C06172=1064.757,412.675,383.902,175.485,36.976,156.989
C06173=1064.765,412.921,383.858,175.491,36.985,156.991
C06174=1064.773,413.167,383.814,175.499,36.994,156.993
C06175=1064.782,413.413,383.769,175.506,37.004,156.996
C06176=1064.790,413.659,383.725,175.512,37.013,156.998
C06177=1064.799,413.905,383.681,175.519,37.023,157.001
C06178=1064.807,414.150,383.637,175.525,37.033,157.003
C06179=1064.817,414.453,383.583,175.534,37.044,157.006
C06180=1064.827,414.756,383.528,175.542,37.056,157.009
C06181=1064.836,415.058,383.473,175.552,37.068,157.012
C06182=1064.847,415.360,383.419,175.560,37.080,157.015
C06183=1064.855,415.607,383.374,175.566,37.090,157.018
C06184=1064.863,415.852,383.330,175.574,37.099,157.020
C06185=1064.872,416.098,383.285,175.581,37.109,157.023
C06186=1064.880,416.343,383.241,175.587,37.119,157.025
C06187=1064.888,416.590,383.195,175.595,37.129,157.028
C06188=1064.896,416.836,383.151,175.602,37.139,157.030
C06189=1064.904,417.081,383.106,175.609,37.149,157.033
C06190=1064.913,417.327,383.061,175.616,37.158,157.035
C06191=1064.921,417.573,383.017,175.623,37.169,157.038
C06192=1064.930,417.819,382.971,175.630,37.179,157.040
C06193=1064.938,418.065,382.927,175.638,37.189,157.043
C06194=1064.946,418.310,382.882,175.644,37.199,157.046
C06195=1064.954,418.557,382.837,175.652,37.209,157.048
C06196=1064.963,418.802,382.792,175.659,37.219,157.051
C06197=1064.971,419.048,382.747,175.666,37.229,157.054
C06198=1064.980,419.293,382.702,175.674,37.239,157.056
C06199=1064.989,419.539,382.656,175.681,37.249,157.059
C06200=1064.997,419.786,382.612,175.688,37.260,157.062
C06201=1065.005,420.031,382.566,175.695,37.270,157.064
C06202=1065.014,420.277,382.521,175.703,37.280,157.067
C06203=1065.022,420.523,382.476,175.710,37.290,157.069
C06204=1065.031,420.768,382.431,175.718,37.301,157.072
C06205=1065.039,421.014,382.385,175.725,37.311,157.075
C06206=1065.048,421.260,382.340,175.733,37.321,157.078
C06207=1065.057,421.505,382.294,175.740,37.332,157.080
C06208=1065.064,421.751,382.249,175.748,37.342,157.083
C06209=1065.073,421.997,382.203,175.756,37.353,157.086
C06210=1065.081,422.243,382.157,175.763,37.363,157.088
C06211=1065.090,422.488,382.112,175.771,37.374,157.091
C06212=1065.098,422.733,382.066,175.778,37.385,157.094
C06213=1065.107,422.979,382.020,175.786,37.395,157.097
C06214=1065.116,423.225,381.975,175.794,37.406,157.100
C06215=1065.124,423.471,381.929,175.801,37.417,157.103
C06216=1065.133,423.716,381.883,175.809,37.427,157.105
C06217=1065.142,423.962,381.837,175.817,37.438,157.108
C06218=1065.151,424.207,381.791,175.824,37.449,157.111
C06219=1065.159,424.453,381.745,175.832,37.459,157.114
C06220=1065.167,424.698,381.700,175.840,37.470,157.117
C06221=1065.176,424.944,381.653,175.848,37.481,157.120
C06222=1065.185,425.190,381.608,175.855,37.492,157.122
C06223=1065.193,425.435,381.561,175.863,37.503,157.125
C06224=1065.203,425.680,381.515,175.871,37.514,157.128
C06225=1065.211,425.927,381.469,175.879,37.525,157.131
C06226=1065.220,426.172,381.423,175.887,37.536,157.134
C06227=1065.229,426.417,381.376,175.895,37.547,157.137
C06228=1065.238,426.662,381.330,175.903,37.558,157.140
C06229=1065.246,426.909,381.284,175.911,37.569,157.143
C06230=1065.255,427.154,381.237,175.919,37.580,157.146
C06231=1065.264,427.399,381.191,175.928,37.592,157.149
C06232=1065.273,427.645,381.144,175.936,37.603,157.152
C06233=1065.281,427.890,381.097,175.943,37.614,157.155
C06234=1065.290,428.136,381.051,175.951,37.626,157.158
C06235=1065.304,428.509,380.979,175.964,37.643,157.163
C06236=1065.317,428.882,380.909,175.976,37.660,157.167
C06237=1065.331,429.255,380.837,175.990,37.678,157.172
C06238=1065.344,429.628,380.766,176.002,37.695,157.177
C06239=1065.353,429.873,380.719,176.011,37.707,157.180
C06240=1065.362,430.118,380.672,176.019,37.718,157.183
C06241=1065.372,430.364,380.626,176.027,37.730,157.186
C06242=1065.381,430.609,380.578,176.036,37.741,157.189
C06243=1065.389,430.855,380.531,176.044,37.753,157.192
C06244=1065.399,431.100,380.484,176.053,37.765,157.195
C06245=1065.407,431.346,380.437,176.061,37.776,157.198
C06246=1065.416,431.591,380.389,176.069,37.788,157.202
C06247=1065.425,431.836,380.342,176.078,37.800,157.205
C06248=1065.434,432.081,380.294,176.086,37.812,157.208
C06249=1065.443,432.327,380.247,176.096,37.824,157.211
C06250=1065.452,432.572,380.200,176.104,37.836,157.215
C06251=1065.461,432.817,380.152,176.113,37.848,157.218
C06252=1065.470,433.062,380.105,176.122,37.861,157.221
C06253=1065.479,433.308,380.057,176.130,37.872,157.224
C06254=1065.488,433.553,380.009,176.140,37.885,157.228
C06255=1065.496,433.772,379.967,176.147,37.896,157.231
C06256=1065.504,433.992,379.923,176.155,37.906,157.234
C06257=1065.512,434.212,379.880,176.163,37.917,157.237
C06258=1065.520,434.432,379.838,176.171,37.928,157.240
C06259=1065.529,434.651,379.796,176.179,37.939,157.243
C06260=1065.538,434.871,379.752,176.187,37.951,157.246
C06261=1065.546,435.091,379.709,176.195,37.961,157.249
C06262=1065.554,435.311,379.666,176.204,37.973,157.252
C06263=1065.564,435.556,379.618,176.212,37.985,157.255
C06264=1065.572,435.801,379.570,176.222,37.997,157.259
C06265=1065.582,436.046,379.522,176.231,38.010,157.262
C06266=1065.591,436.292,379.473,176.239,38.022,157.265
C06267=1065.600,436.536,379.425,176.249,38.035,157.269
C06268=1065.610,436.782,379.377,176.258,38.047,157.272
C06269=1065.619,437.027,379.329,176.268,38.060,157.276
C06270=1065.629,437.272,379.280,176.277,38.073,157.279
C06271=1065.638,437.518,379.233,176.287,38.086,157.283
C06272=1065.648,437.762,379.184,176.295,38.099,157.287
C06273=1065.657,438.007,379.135,176.305,38.111,157.290
C06274=1065.666,438.252,379.087,176.315,38.124,157.294
C06275=1065.676,438.497,379.038,176.324,38.137,157.297
C06276=1065.685,438.742,378.989,176.334,38.150,157.301
C06277=1065.695,438.987,378.941,176.343,38.163,157.304
C06278=1065.705,439.232,378.892,176.353,38.176,157.308
C06279=1065.714,439.478,378.843,176.363,38.189,157.312
C06280=1065.724,439.722,378.794,176.372,38.202,157.315
C06281=1065.733,439.967,378.746,176.382,38.215,157.319
C06282=1065.743,440.212,378.696,176.392,38.229,157.323
C06283=1065.752,440.457,378.648,176.401,38.242,157.326
C06284=1065.761,440.702,378.598,176.411,38.255,157.330
C06285=1065.771,440.947,378.549,176.421,38.269,157.334
C06286=1065.780,441.192,378.500,176.431,38.282,157.338
C06287=1065.791,441.436,378.451,176.440,38.295,157.341
C06288=1065.800,441.682,378.402,176.451,38.309,157.345
C06289=1065.810,441.926,378.352,176.461,38.322,157.349
C06290=1065.819,442.171,378.303,176.471,38.336,157.353
C06291=1065.828,442.394,378.257,176.480,38.348,157.356
C06292=1065.836,442.618,378.212,176.489,38.361,157.360
C06293=1065.846,442.841,378.168,176.499,38.373,157.363
C06294=1065.855,443.065,378.122,176.508,38.386,157.367
C06295=1065.864,443.288,378.077,176.517,38.398,157.371
C06296=1065.873,443.512,378.031,176.527,38.411,157.374
C06297=1065.881,443.735,377.986,176.536,38.424,157.378
C06298=1065.890,443.959,377.941,176.546,38.436,157.381
C06299=1065.900,444.204,377.890,176.556,38.450,157.385
C06300=1065.910,444.448,377.841,176.567,38.464,157.389
C06301=1065.920,444.692,377.791,176.577,38.478,157.393
C06302=1065.930,444.938,377.740,176.587,38.492,157.397
C06303=1065.939,445.182,377.691,176.598,38.506,157.401
C06304=1065.950,445.427,377.640,176.608,38.520,157.405
C06305=1065.960,445.671,377.590,176.619,38.535,157.409
C06306=1065.969,445.917,377.540,176.629,38.549,157.413
C06307=1065.980,446.160,377.490,176.640,38.564,157.418
C06308=1065.990,446.405,377.439,176.652,38.578,157.422
C06309=1065.999,446.650,377.390,176.662,38.592,157.426
C06310=1066.010,446.895,377.339,176.673,38.607,157.430
C06311=1066.020,447.138,377.289,176.683,38.621,157.434
C06312=1066.030,447.383,377.238,176.695,38.636,157.438
C06313=1066.040,447.627,377.187,176.706,38.650,157.443
C06314=1066.051,447.872,377.137,176.716,38.665,157.447
C06315=1066.062,448.115,377.088,176.728,38.679,157.451
C06316=1066.074,448.359,377.038,176.739,38.693,157.455
C06317=1066.087,448.603,376.991,176.750,38.707,157.459
C06318=1066.101,448.848,376.942,176.761,38.720,157.463
C06319=1066.118,449.093,376.895,176.773,38.733,157.467
C06320=1066.134,449.338,376.849,176.783,38.746,157.470
C06321=1066.151,449.584,376.803,176.794,38.758,157.474
C06322=1066.169,449.829,376.758,176.804,38.770,157.477
C06323=1065.829,449.834,376.494,176.795,38.897,157.512
C06324=1065.810,449.588,376.540,176.785,38.885,157.508
C06325=1065.792,449.342,376.585,176.773,38.873,157.505
C06326=1065.776,449.097,376.631,176.763,38.861,157.501
C06327=1065.760,448.852,376.679,176.752,38.848,157.497
C06328=1065.746,448.608,376.726,176.740,38.834,157.493
C06329=1065.733,448.363,376.774,176.729,38.821,157.489
C06330=1065.720,448.119,376.824,176.717,38.807,157.485
C06331=1065.708,447.876,376.872,176.706,38.793,157.481
C06332=1065.698,447.631,376.923,176.694,38.778,157.477
C06333=1065.687,447.388,376.974,176.684,38.764,157.473
C06334=1065.677,447.143,377.025,176.673,38.750,157.469
C06335=1065.668,446.899,377.075,176.661,38.735,157.464
C06336=1065.657,446.654,377.125,176.651,38.721,157.460
C06337=1065.647,446.410,377.176,176.640,38.706,157.456
C06338=1065.637,446.166,377.227,176.629,38.692,157.452
C06339=1065.627,445.921,377.276,176.618,38.677,157.448
C06340=1065.617,445.677,377.327,176.607,38.663,157.444
C06341=1065.607,445.431,377.377,176.597,38.649,157.440
C06342=1065.597,445.187,377.427,176.586,38.635,157.436
C06343=1065.586,444.942,377.477,176.575,38.621,157.432
C06344=1065.577,444.697,377.527,176.565,38.607,157.427
C06345=1065.568,444.453,377.577,176.554,38.593,157.423
C06346=1065.557,444.208,377.627,176.544,38.579,157.419
C06347=1065.548,443.964,377.677,176.534,38.565,157.416
C06348=1065.538,443.750,377.721,176.523,38.553,157.412
C06349=1065.530,443.536,377.764,176.515,38.541,157.409
C06350=1065.522,443.322,377.808,176.506,38.529,157.405
C06351=1065.513,443.108,377.851,176.497,38.517,157.402
C06352=1065.504,442.894,377.894,176.488,38.505,157.398
C06353=1065.496,442.680,377.937,176.479,38.493,157.395
C06354=1065.487,442.467,377.981,176.470,38.481,157.391
C06355=1065.478,442.252,378.024,176.461,38.469,157.388
C06356=1065.469,442.008,378.074,176.451,38.456,157.384
C06357=1065.459,441.763,378.123,176.441,38.442,157.380
C06358=1065.450,441.518,378.173,176.430,38.429,157.377
C06359=1065.440,441.274,378.222,176.421,38.415,157.373
C06360=1065.431,441.028,378.271,176.411,38.402,157.369
C06361=1065.420,440.783,378.321,176.401,38.388,157.365
C06362=1065.411,440.538,378.370,176.391,38.375,157.362
C06363=1065.401,440.294,378.419,176.380,38.362,157.358
C06364=1065.392,440.048,378.468,176.371,38.349,157.354
C06365=1065.382,439.803,378.517,176.361,38.335,157.350
C06366=1065.372,439.559,378.566,176.351,38.323,157.347
C06367=1065.363,439.314,378.615,176.342,38.309,157.343
C06368=1065.353,439.069,378.663,176.332,38.296,157.339
C06369=1065.344,438.823,378.713,176.322,38.284,157.336
C06370=1065.335,438.578,378.761,176.313,38.270,157.332
C06371=1065.326,438.334,378.809,176.303,38.258,157.329
C06372=1065.317,438.089,378.858,176.294,38.245,157.325
C06373=1065.307,437.844,378.907,176.284,38.232,157.322
C06374=1065.297,437.599,378.955,176.274,38.219,157.318
C06375=1065.287,437.354,379.004,176.265,38.206,157.314
C06376=1065.277,437.109,379.053,176.255,38.194,157.311
C06377=1065.268,436.863,379.100,176.246,38.181,157.307
C06378=1065.259,436.618,379.149,176.237,38.169,157.304
C06379=1065.250,436.374,379.198,176.228,38.156,157.300
C06380=1065.240,436.128,379.245,176.218,38.144,157.297
C06381=1065.231,435.883,379.294,176.209,38.131,157.294
C06382=1065.221,435.638,379.342,176.200,38.118,157.290
C06383=1065.212,435.393,379.390,176.191,38.106,157.287
C06384=1065.203,435.148,379.438,176.182,38.094,157.283
C06385=1065.194,434.903,379.485,176.172,38.082,157.280
C06386=1065.185,434.658,379.534,176.163,38.069,157.276
C06387=1065.175,434.412,379.582,176.155,38.057,157.273
C06388=1065.166,434.167,379.630,176.145,38.045,157.270
C06389=1065.157,433.922,379.677,176.136,38.033,157.266
C06390=1065.148,433.677,379.726,176.128,38.021,157.263
C06391=1065.138,433.432,379.773,176.119,38.008,157.260
C06392=1065.129,433.187,379.821,176.109,37.996,157.256
C06393=1065.120,432.941,379.869,176.101,37.985,157.253
C06394=1065.111,432.696,379.916,176.092,37.972,157.250
C06395=1065.102,432.451,379.964,176.084,37.960,157.247
C06396=1065.093,432.206,380.011,176.075,37.948,157.243
C06397=1065.084,431.960,380.058,176.066,37.937,157.240
C06398=1065.075,431.715,380.106,176.057,37.925,157.237
C06399=1065.066,431.470,380.153,176.048,37.913,157.234
C06400=1065.057,431.225,380.201,176.040,37.901,157.230
C06401=1065.048,430.979,380.248,176.031,37.889,157.227
C06402=1065.039,430.734,380.295,176.023,37.878,157.224
C06403=1065.030,430.488,380.342,176.015,37.866,157.221
C06404=1065.021,430.243,380.390,176.006,37.854,157.218
C06405=1065.012,429.998,380.436,175.998,37.843,157.215
C06406=1065.003,429.753,380.483,175.989,37.831,157.212
C06407=1064.994,429.506,380.530,175.981,37.820,157.209
C06408=1064.982,429.183,380.592,175.970,37.804,157.204
C06409=1064.971,428.859,380.654,175.959,37.789,157.200
C06410=1064.958,428.535,380.716,175.947,37.774,157.196
C06411=1064.947,428.210,380.778,175.936,37.759,157.192
C06412=1064.938,427.965,380.824,175.928,37.748,157.189
C06413=1064.930,427.720,380.871,175.920,37.737,157.186
C06414=1064.921,427.475,380.918,175.911,37.725,157.183
C06415=1064.912,427.229,380.965,175.903,37.715,157.180
C06416=1064.903,426.984,381.011,175.896,37.703,157.177
C06417=1064.894,426.737,381.057,175.888,37.692,157.174
C06418=1064.886,426.492,381.104,175.879,37.681,157.171
C06419=1064.876,426.247,381.150,175.871,37.670,157.168
C06420=1064.868,426.001,381.197,175.863,37.659,157.165
C06421=1064.858,425.756,381.243,175.855,37.648,157.162
C06422=1064.850,425.510,381.289,175.848,37.637,157.160
C06423=1064.841,425.265,381.335,175.839,37.626,157.157
C06424=1064.830,424.958,381.393,175.830,37.612,157.153
C06425=1064.820,424.652,381.450,175.819,37.599,157.149
C06426=1064.809,424.345,381.507,175.809,37.585,157.146
C06427=1064.798,424.038,381.565,175.800,37.572,157.142
C06428=1064.788,423.793,381.611,175.792,37.561,157.139
C06429=1064.780,423.547,381.657,175.785,37.551,157.137
C06430=1064.772,423.302,381.702,175.776,37.540,157.134
C06431=1064.763,423.056,381.749,175.768,37.529,157.131
C06432=1064.754,422.810,381.794,175.761,37.519,157.128
C06433=1064.746,422.564,381.840,175.753,37.509,157.125
C06434=1064.738,422.319,381.885,175.746,37.498,157.123
C06435=1064.729,422.073,381.932,175.738,37.487,157.120
C06436=1064.720,421.828,381.978,175.730,37.477,157.117
C06437=1064.712,421.583,382.023,175.723,37.466,157.114
C06438=1064.704,421.336,382.069,175.715,37.456,157.112
C06439=1064.695,421.091,382.114,175.708,37.445,157.109
C06440=1064.687,420.845,382.160,175.700,37.435,157.106
C06441=1064.678,420.599,382.205,175.693,37.425,157.103
C06442=1064.669,420.354,382.250,175.685,37.414,157.101
C06443=1064.661,420.108,382.295,175.678,37.404,157.098
C06444=1064.653,419.862,382.341,175.671,37.394,157.095
C06445=1064.644,419.616,382.386,175.664,37.384,157.093
C06446=1064.635,419.371,382.431,175.656,37.374,157.090
C06447=1064.627,419.124,382.476,175.649,37.364,157.088
C06448=1064.618,418.879,382.521,175.641,37.353,157.085
C06449=1064.609,418.633,382.566,175.634,37.343,157.082
C06450=1064.602,418.387,382.611,175.626,37.333,157.080
C06451=1064.593,418.141,382.657,175.619,37.323,157.077
C06452=1064.585,417.896,382.701,175.612,37.313,157.074
C06453=1064.576,417.650,382.747,175.605,37.303,157.072
C06454=1064.568,417.404,382.791,175.598,37.293,157.069
C06455=1064.560,417.159,382.836,175.590,37.284,157.067
C06456=1064.551,416.913,382.881,175.583,37.274,157.064
C06457=1064.543,416.667,382.925,175.577,37.264,157.062
C06458=1064.535,416.421,382.971,175.569,37.254,157.059
C06459=1064.526,416.175,383.015,175.562,37.244,157.056
C06460=1064.518,415.931,383.059,175.555,37.234,157.054
C06461=1064.510,415.686,383.104,175.549,37.224,157.051
C06462=1064.502,415.442,383.148,175.541,37.215,157.049
C06463=1064.494,415.197,383.193,175.534,37.205,157.047
C06464=1064.485,414.952,383.237,175.527,37.196,157.044
C06465=1064.477,414.708,383.281,175.521,37.186,157.041
C06466=1064.469,414.463,383.325,175.513,37.176,157.039
C06467=1064.461,414.219,383.369,175.506,37.167,157.037
C06468=1064.452,413.974,383.413,175.500,37.157,157.034
C06469=1064.444,413.727,383.458,175.493,37.148,157.032
C06470=1064.436,413.481,383.502,175.486,37.139,157.029
C06471=1064.428,413.235,383.546,175.479,37.129,157.027
C06472=1064.419,412.990,383.590,175.472,37.120,157.024
C06473=1064.411,412.744,383.634,175.465,37.111,157.022
C06474=1064.403,412.498,383.678,175.459,37.101,157.020
C06475=1064.395,412.251,383.722,175.452,37.091,157.017
C06476=1064.386,412.006,383.766,175.446,37.082,157.015
C06477=1064.378,411.760,383.810,175.438,37.073,157.013
C06478=1064.370,411.513,383.854,175.431,37.064,157.010
C06479=1064.362,411.268,383.898,175.425,37.055,157.008
C06480=1064.353,411.022,383.941,175.418,37.045,157.006
C06481=1064.345,410.776,383.986,175.412,37.036,157.003
C06482=1064.338,410.530,384.029,175.405,37.027,157.001
C06483=1064.330,410.283,384.073,175.399,37.018,156.999
C06484=1064.321,410.038,384.117,175.392,37.008,156.996
C06485=1064.313,409.791,384.160,175.385,36.999,156.994
C06486=1064.305,409.546,384.205,175.379,36.990,156.992
C06487=1064.297,409.300,384.248,175.372,36.981,156.989
C06488=1064.289,409.053,384.291,175.366,36.972,156.987
C06489=1064.281,408.807,384.335,175.359,36.963,156.985
C06490=1064.273,408.561,384.378,175.353,36.955,156.983
C06491=1064.265,408.315,384.422,175.346,36.945,156.980
C06492=1064.257,408.069,384.465,175.340,36.936,156.978
C06493=1064.249,407.823,384.508,175.333,36.927,156.976
C06494=1064.241,407.577,384.552,175.327,36.919,156.974
C06495=1064.233,407.331,384.596,175.321,36.910,156.971
C06496=1064.225,407.085,384.639,175.314,36.901,156.969
C06497=1064.218,406.839,384.682,175.308,36.892,156.967
C06498=1064.210,406.593,384.726,175.301,36.883,156.964
C06499=1064.201,406.346,384.769,175.296,36.874,156.962
C06500=1064.194,406.100,384.812,175.289,36.866,156.960
C06501=1064.186,405.854,384.854,175.283,36.857,156.958
C06502=1064.178,405.608,384.898,175.276,36.848,156.956
C06503=1064.170,405.362,384.941,175.270,36.839,156.954
C06504=1064.163,405.116,384.984,175.264,36.831,156.951
C06505=1064.155,404.869,385.026,175.257,36.822,156.949
C06506=1064.147,404.623,385.070,175.252,36.814,156.947
C06507=1064.139,404.378,385.113,175.246,36.805,156.945
C06508=1064.131,404.131,385.156,175.239,36.797,156.943
C06509=1064.123,403.885,385.199,175.233,36.788,156.941
C06510=1064.115,403.639,385.241,175.227,36.779,156.939
C06511=1064.108,403.392,385.284,175.220,36.771,156.936
C06512=1064.099,403.146,385.327,175.215,36.762,156.934
C06513=1064.091,402.900,385.369,175.209,36.754,156.932
C06514=1064.084,402.653,385.412,175.202,36.745,156.930
C06515=1064.076,402.408,385.455,175.196,36.737,156.928
C06516=1064.068,402.161,385.497,175.191,36.729,156.926
C06517=1064.061,401.915,385.540,175.184,36.721,156.924
C06518=1064.053,401.668,385.582,175.178,36.712,156.922
C06519=1064.045,401.423,385.625,175.172,36.704,156.920
C06520=1064.035,401.123,385.676,175.165,36.694,156.917
C06521=1064.026,400.823,385.727,175.158,36.684,156.915
C06522=1064.017,400.524,385.779,175.150,36.674,156.912
C06523=1064.007,400.225,385.830,175.144,36.664,156.910
C06524=1063.999,399.978,385.873,175.137,36.655,156.908
C06525=1063.991,399.732,385.915,175.131,36.647,156.906
C06526=1063.984,399.486,385.957,175.126,36.639,156.904
C06527=1063.976,399.239,385.999,175.120,36.631,156.902
C06528=1063.969,398.993,386.042,175.113,36.623,156.900
C06529=1063.961,398.747,386.083,175.108,36.615,156.898
C06530=1063.953,398.500,386.126,175.102,36.607,156.896
C06531=1063.945,398.254,386.168,175.096,36.599,156.894
C06532=1063.938,398.008,386.210,175.091,36.591,156.892
C06533=1063.930,397.762,386.252,175.084,36.583,156.890
C06534=1063.922,397.515,386.293,175.079,36.575,156.888
C06535=1063.915,397.269,386.335,175.073,36.567,156.886
C06536=1063.907,397.023,386.377,175.067,36.559,156.884
C06537=1063.899,396.777,386.419,175.062,36.551,156.882
C06538=1063.892,396.530,386.461,175.056,36.544,156.880
C06539=1063.884,396.284,386.503,175.050,36.535,156.878
C06540=1063.876,396.038,386.545,175.044,36.528,156.877
C06541=1063.869,395.791,386.586,175.039,36.520,156.875
C06542=1063.862,395.545,386.628,175.033,36.512,156.873
C06543=1063.854,395.298,386.669,175.027,36.504,156.871
C06544=1063.846,395.052,386.711,175.022,36.496,156.869
C06545=1063.839,394.806,386.752,175.016,36.489,156.867
C06546=1063.831,394.560,386.794,175.011,36.481,156.865
C06547=1063.823,394.313,386.835,175.004,36.473,156.863
C06548=1063.816,394.067,386.876,174.999,36.465,156.861
C06549=1063.808,393.821,386.918,174.993,36.458,156.859
C06550=1063.801,393.574,386.959,174.988,36.450,156.858
C06551=1063.793,393.328,387.001,174.982,36.442,156.856
C06552=1063.786,393.082,387.043,174.977,36.435,156.854
C06553=1063.778,392.835,387.083,174.971,36.427,156.852
C06554=1063.771,392.589,387.125,174.966,36.420,156.850
C06555=1063.764,392.342,387.166,174.960,36.412,156.848
C06556=1063.756,392.096,387.208,174.955,36.404,156.847
C06557=1063.748,391.850,387.248,174.950,36.397,156.845
C06558=1063.741,391.603,387.290,174.944,36.390,156.843
C06559=1063.733,391.357,387.331,174.939,36.382,156.841
C06560=1063.725,391.110,387.371,174.932,36.374,156.839
C06561=1063.718,390.864,387.413,174.927,36.367,156.838
C06562=1063.711,390.617,387.454,174.921,36.360,156.836
C06563=1063.703,390.371,387.495,174.916,36.353,156.834
C06564=1063.695,390.124,387.536,174.911,36.345,156.832
C06565=1063.688,389.879,387.576,174.905,36.338,156.831
C06566=1063.681,389.632,387.617,174.900,36.330,156.829
C06567=1063.673,389.386,387.658,174.894,36.323,156.827
C06568=1063.666,389.139,387.698,174.889,36.316,156.825
C06569=1063.658,388.892,387.739,174.884,36.308,156.823
C06570=1063.650,388.646,387.780,174.878,36.301,156.822
C06571=1063.642,388.399,387.821,174.873,36.294,156.820
C06572=1063.635,388.152,387.861,174.867,36.287,156.818
C06573=1063.628,387.907,387.902,174.863,36.280,156.817
C06574=1063.621,387.660,387.943,174.857,36.272,156.815
C06575=1063.613,387.413,387.983,174.852,36.265,156.813
C06576=1063.605,387.131,388.030,174.845,36.257,156.811
C06577=1063.596,386.848,388.076,174.839,36.249,156.809
C06578=1063.588,386.565,388.122,174.834,36.240,156.807
C06579=1063.579,386.282,388.169,174.828,36.233,156.805
C06580=1063.571,386.035,388.209,174.822,36.226,156.804
C06581=1063.565,385.789,388.250,174.817,36.218,156.802
C06582=1063.557,385.542,388.290,174.812,36.211,156.800
C06583=1063.549,385.295,388.330,174.806,36.204,156.799
C06584=1063.542,385.049,388.371,174.802,36.197,156.797
C06585=1063.535,384.802,388.411,174.797,36.190,156.795
C06586=1063.528,384.556,388.451,174.792,36.183,156.794
C06587=1063.520,384.310,388.492,174.786,36.176,156.792
C06588=1063.513,384.063,388.531,174.781,36.169,156.790
C06589=1063.506,383.816,388.572,174.776,36.162,156.789
C06590=1063.498,383.570,388.612,174.771,36.155,156.787
C06591=1063.491,383.324,388.652,174.765,36.148,156.785
C06592=1063.484,383.077,388.692,174.760,36.141,156.784
C06593=1063.476,382.830,388.732,174.755,36.134,156.782
C06594=1063.470,382.583,388.772,174.751,36.128,156.780
C06595=1063.463,382.337,388.812,174.746,36.121,156.779
C06596=1063.455,382.090,388.852,174.740,36.114,156.777
C06597=1063.448,381.843,388.892,174.735,36.107,156.775
C06598=1063.441,381.597,388.932,174.730,36.100,156.774
C06599=1063.434,381.350,388.971,174.725,36.093,156.772
C06600=1063.427,381.103,389.012,174.720,36.086,156.771
C06601=1063.420,380.857,389.052,174.716,36.080,156.769
C06602=1063.412,380.610,389.091,174.710,36.073,156.768
C06603=1063.405,380.364,389.131,174.705,36.066,156.766
C06604=1063.397,380.117,389.171,174.700,36.059,156.764
C06605=1063.390,379.871,389.210,174.695,36.053,156.763
C06606=1063.383,379.623,389.250,174.690,36.046,156.761
C06607=1063.376,379.377,389.289,174.685,36.039,156.760
C06608=1063.368,379.130,389.329,174.680,36.033,156.758
C06609=1063.361,378.884,389.369,174.675,36.026,156.757
C06610=1063.353,378.636,389.408,174.670,36.019,156.755
C06611=1063.346,378.390,389.447,174.665,36.013,156.753
C06612=1063.339,378.144,389.487,174.660,36.006,156.752
C06613=1063.332,377.896,389.526,174.656,36.000,156.750
C06614=1063.325,377.650,389.566,174.651,35.993,156.749
C06615=1063.318,377.403,389.605,174.646,35.987,156.747
C06616=1063.310,377.157,389.644,174.640,35.980,156.746
C06617=1063.303,376.910,389.683,174.635,35.973,156.744
C06618=1063.296,376.663,389.723,174.631,35.967,156.743
C06619=1063.289,376.416,389.762,174.626,35.961,156.741
C06620=1063.282,376.170,389.802,174.621,35.954,156.740
C06621=1063.275,375.923,389.840,174.616,35.947,156.738
C06622=1063.267,375.676,389.880,174.612,35.941,156.737
C06623=1063.260,375.429,389.919,174.607,35.935,156.735
C06624=1063.253,375.182,389.958,174.602,35.929,156.734
C06625=1063.246,374.936,389.998,174.597,35.922,156.732
C06626=1063.240,374.689,390.036,174.593,35.915,156.731
C06627=1063.232,374.442,390.076,174.588,35.909,156.729
C06628=1063.225,374.195,390.115,174.583,35.902,156.728
C06629=1063.218,373.949,390.154,174.578,35.896,156.726
C06630=1063.211,373.702,390.193,174.574,35.890,156.725
C06631=1063.205,373.455,390.232,174.569,35.884,156.723
C06632=1063.197,373.203,390.272,174.564,35.877,156.722
C06633=1063.190,372.951,390.312,174.559,35.871,156.720
C06634=1063.183,372.699,390.351,174.555,35.864,156.719
C06635=1063.175,372.446,390.391,174.550,35.858,156.717
C06636=1063.168,372.200,390.430,174.545,35.851,156.716
C06637=1063.161,371.953,390.468,174.540,35.845,156.714
C06638=1063.154,371.706,390.507,174.536,35.839,156.713
C06639=1063.147,371.460,390.545,174.531,35.833,156.712
C06640=1063.140,371.213,390.584,174.526,35.827,156.710
C06641=1063.133,370.965,390.623,174.522,35.821,156.709
C06642=1063.125,370.718,390.661,174.517,35.814,156.707
C06643=1063.118,370.471,390.700,174.512,35.808,156.706
C06644=1063.111,370.225,390.738,174.507,35.802,156.705
C06645=1063.104,369.978,390.777,174.503,35.796,156.703
C06646=1063.097,369.731,390.816,174.498,35.790,156.702
C06647=1063.090,369.484,390.853,174.493,35.784,156.700
C06648=1063.083,369.237,390.892,174.489,35.778,156.699
C06649=1063.076,368.990,390.931,174.484,35.771,156.698
C06650=1063.069,368.743,390.968,174.479,35.765,156.696
C06651=1063.062,368.496,391.007,174.475,35.759,156.695
C06652=1063.055,368.250,391.046,174.470,35.754,156.693
C06653=1063.048,368.002,391.084,174.466,35.747,156.692
C06654=1063.042,367.756,391.123,174.462,35.741,156.691
C06655=1063.034,367.509,391.161,174.457,35.735,156.689
C06656=1063.027,367.262,391.199,174.452,35.729,156.688
C06657=1063.020,367.015,391.237,174.448,35.723,156.687
C06658=1063.013,366.768,391.275,174.443,35.717,156.685
C06659=1063.006,366.521,391.314,174.438,35.711,156.684
C06660=1062.999,366.274,391.352,174.434,35.705,156.682
C06661=1062.993,366.027,391.390,174.430,35.699,156.681
C06662=1062.986,365.780,391.428,174.425,35.694,156.680
C06663=1062.979,365.533,391.466,174.421,35.687,156.678
C06664=1062.972,365.286,391.504,174.416,35.681,156.677
C06665=1062.965,365.039,391.542,174.412,35.676,156.676
C06666=1062.958,364.793,391.580,174.407,35.669,156.674
C06667=1062.951,364.545,391.618,174.403,35.664,156.673
C06668=1062.945,364.299,391.656,174.399,35.658,156.672
C06669=1062.938,364.051,391.694,174.394,35.652,156.670
C06670=1062.931,363.805,391.732,174.389,35.646,156.669
C06671=1062.924,363.557,391.770,174.385,35.640,156.668
C06672=1062.917,363.310,391.808,174.380,35.635,156.666
C06673=1062.910,363.063,391.845,174.377,35.628,156.665
C06674=1062.903,362.815,391.883,174.372,35.623,156.664
C06675=1062.896,362.569,391.920,174.367,35.617,156.662
C06676=1062.889,362.322,391.958,174.363,35.612,156.661
C06677=1062.882,362.075,391.996,174.358,35.605,156.660
C06678=1062.875,361.828,392.034,174.355,35.600,156.658
C06679=1062.868,361.582,392.072,174.350,35.594,156.657
C06680=1062.861,361.334,392.109,174.345,35.588,156.656
C06681=1062.854,361.087,392.146,174.341,35.583,156.655
C06682=1062.848,360.839,392.184,174.337,35.577,156.653
C06683=1062.841,360.593,392.221,174.333,35.572,156.652
C06684=1062.834,360.352,392.258,174.328,35.566,156.651
C06685=1062.827,360.112,392.295,174.323,35.560,156.650
C06686=1062.821,359.871,392.331,174.320,35.555,156.648
C06687=1062.814,359.630,392.367,174.315,35.549,156.647
C06688=1062.807,359.389,392.404,174.312,35.544,156.646
C06689=1062.801,359.149,392.440,174.307,35.538,156.645
C06690=1062.794,358.908,392.476,174.303,35.533,156.643
C06691=1062.788,358.668,392.513,174.299,35.528,156.642
C06692=1062.781,358.421,392.550,174.295,35.522,156.641
C06693=1062.773,358.173,392.588,174.290,35.516,156.640
C06694=1062.767,357.926,392.624,174.285,35.511,156.638
C06695=1062.760,357.679,392.662,174.282,35.505,156.637
C06696=1062.753,357.432,392.699,174.277,35.499,156.636
C06697=1062.746,357.185,392.736,174.273,35.494,156.635
C06698=1062.739,356.938,392.773,174.269,35.489,156.633
C06699=1062.732,356.691,392.810,174.265,35.483,156.632
C06700=1062.726,356.444,392.847,174.260,35.477,156.631
C06701=1062.718,356.197,392.885,174.257,35.472,156.630
C06702=1062.712,355.949,392.921,174.252,35.466,156.629
C06703=1062.705,355.702,392.959,174.248,35.461,156.627
C06704=1062.698,355.455,392.995,174.244,35.456,156.626
C06705=1062.691,355.208,393.032,174.240,35.450,156.625
C06706=1062.685,354.961,393.069,174.235,35.444,156.624
C06707=1062.678,354.713,393.106,174.231,35.439,156.622
C06708=1062.671,354.467,393.143,174.227,35.434,156.621
C06709=1062.664,354.219,393.180,174.222,35.428,156.620
C06710=1062.658,353.972,393.216,174.219,35.423,156.619
C06711=1062.651,353.725,393.254,174.214,35.417,156.618
C06712=1062.644,353.478,393.290,174.210,35.412,156.616
C06713=1062.637,353.230,393.327,174.206,35.406,156.615
C06714=1062.631,352.984,393.364,174.202,35.401,156.614
C06715=1062.624,352.736,393.401,174.198,35.396,156.613
C06716=1062.617,352.489,393.438,174.194,35.390,156.612
C06717=1062.611,352.241,393.474,174.189,35.385,156.611
C06718=1062.604,351.994,393.511,174.186,35.380,156.609
C06719=1062.598,351.747,393.547,174.181,35.374,156.608
C06720=1062.591,351.500,393.585,174.178,35.369,156.607
C06721=1062.584,351.253,393.621,174.173,35.364,156.606
C06722=1062.577,351.005,393.657,174.169,35.359,156.605
C06723=1062.570,350.758,393.694,174.165,35.353,156.603
C06724=1062.563,350.511,393.731,174.161,35.348,156.602
C06725=1062.556,350.264,393.767,174.157,35.343,156.601
C06726=1062.550,350.017,393.803,174.153,35.338,156.600
C06727=1062.543,349.769,393.840,174.148,35.332,156.599
C06728=1062.537,349.522,393.876,174.145,35.327,156.598
C06729=1062.530,349.275,393.912,174.140,35.322,156.596
C06730=1062.523,349.028,393.949,174.137,35.316,156.595
C06731=1062.517,348.780,393.985,174.132,35.311,156.594
C06732=1062.510,348.533,394.021,174.129,35.306,156.593
C06733=1062.503,348.285,394.057,174.125,35.301,156.592
C06734=1062.496,348.038,394.094,174.121,35.295,156.591
C06735=1062.490,347.791,394.130,174.117,35.290,156.590
C06736=1062.482,347.544,394.166,174.112,35.285,156.588
C06737=1062.476,347.296,394.202,174.109,35.280,156.587
C06738=1062.470,347.049,394.239,174.104,35.275,156.586
C06739=1062.463,346.802,394.274,174.101,35.270,156.585
C06740=1062.456,346.563,394.309,174.097,35.265,156.584
C06741=1062.450,346.325,394.344,174.093,35.260,156.583
C06742=1062.444,346.086,394.379,174.089,35.255,156.582
C06743=1062.437,345.848,394.414,174.085,35.250,156.581
C06744=1062.430,345.610,394.448,174.082,35.245,156.580
C06745=1062.425,345.371,394.483,174.078,35.240,156.579
C06746=1062.418,345.132,394.518,174.074,35.235,156.578
C06747=1062.412,344.894,394.552,174.070,35.230,156.576
C06748=1062.405,344.647,394.589,174.066,35.225,156.575
C06749=1062.398,344.399,394.624,174.062,35.220,156.574
C06750=1062.392,344.152,394.661,174.058,35.215,156.573
C06751=1062.385,343.904,394.696,174.055,35.210,156.572
C06752=1062.378,343.657,394.732,174.051,35.205,156.571
C06753=1062.372,343.410,394.767,174.047,35.200,156.570
C06754=1062.366,343.162,394.803,174.043,35.195,156.569
C06755=1062.358,342.915,394.839,174.039,35.189,156.568
C06756=1062.352,342.667,394.875,174.035,35.185,156.567
C06757=1062.345,342.420,394.911,174.031,35.180,156.565
C06758=1062.338,342.173,394.946,174.027,35.175,156.564
C06759=1062.332,341.925,394.982,174.023,35.170,156.563
C06760=1062.325,341.679,395.018,174.020,35.165,156.562
C06761=1062.318,341.431,395.053,174.015,35.160,156.561
C06762=1062.312,341.183,395.089,174.012,35.155,156.560
C06763=1062.305,340.935,395.124,174.008,35.150,156.559
C06764=1062.298,340.688,395.159,174.004,35.145,156.558
C06765=1062.292,340.441,395.196,174.001,35.140,156.557
C06766=1062.285,340.194,395.231,173.996,35.135,156.556
C06767=1062.278,339.946,395.266,173.993,35.130,156.555
C06768=1062.272,339.699,395.302,173.989,35.125,156.554
C06769=1062.265,339.451,395.337,173.985,35.121,156.553
C06770=1062.259,339.204,395.372,173.981,35.115,156.552
C06771=1062.253,338.956,395.408,173.977,35.111,156.551
C06772=1062.245,338.709,395.444,173.974,35.106,156.549
C06773=1062.239,338.462,395.479,173.970,35.101,156.548
C06774=1062.233,338.214,395.514,173.966,35.096,156.547
C06775=1062.226,337.967,395.550,173.963,35.091,156.546
C06776=1062.219,337.720,395.585,173.958,35.086,156.545
C06777=1062.213,337.472,395.620,173.955,35.081,156.544
C06778=1062.206,337.225,395.656,173.951,35.076,156.543
C06779=1062.200,336.977,395.691,173.947,35.072,156.542
C06780=1062.193,336.729,395.725,173.944,35.067,156.541
C06781=1062.186,336.482,395.760,173.940,35.062,156.540
C06782=1062.180,336.235,395.795,173.936,35.057,156.539
C06783=1062.174,335.987,395.831,173.932,35.053,156.538
C06784=1062.167,335.740,395.866,173.929,35.047,156.537
C06785=1062.161,335.493,395.901,173.925,35.043,156.536
C06786=1062.154,335.245,395.935,173.921,35.038,156.535
C06787=1062.147,334.997,395.971,173.918,35.034,156.534
C06788=1062.141,334.750,396.006,173.913,35.028,156.533
C06789=1062.134,334.503,396.041,173.910,35.024,156.532
C06790=1062.127,334.255,396.075,173.907,35.019,156.531
C06791=1062.121,334.007,396.110,173.902,35.014,156.530
C06792=1062.114,333.760,396.145,173.899,35.009,156.529
C06793=1062.108,333.513,396.180,173.896,35.005,156.528
C06794=1062.101,333.265,396.215,173.891,35.000,156.527
C06795=1062.094,333.018,396.250,173.888,34.995,156.526
C06796=1062.088,332.777,396.284,173.885,34.991,156.525
C06797=1062.082,332.536,396.317,173.881,34.986,156.524
C06798=1062.076,332.295,396.352,173.877,34.981,156.523
C06799=1062.069,332.054,396.385,173.874,34.977,156.522
C06800=1062.063,331.814,396.419,173.870,34.972,156.521
C06801=1062.056,331.573,396.453,173.867,34.968,156.520
C06802=1062.050,331.331,396.487,173.863,34.963,156.519
C06803=1062.044,331.091,396.520,173.860,34.958,156.518
C06804=1062.037,330.843,396.555,173.856,34.954,156.517
C06805=1062.031,330.595,396.589,173.852,34.949,156.516
C06806=1062.025,330.348,396.624,173.849,34.944,156.515
C06807=1062.018,330.100,396.658,173.845,34.940,156.514
C06808=1062.011,329.853,396.692,173.841,34.936,156.513
C06809=1062.004,329.605,396.727,173.838,34.931,156.512
C06810=1061.998,329.357,396.762,173.835,34.926,156.511
C06811=1061.991,329.110,396.796,173.830,34.922,156.510
C06812=1061.985,328.863,396.830,173.827,34.917,156.509
C06813=1061.978,328.615,396.865,173.824,34.913,156.508
C06814=1061.971,328.367,396.899,173.820,34.908,156.507
C06815=1061.964,328.119,396.933,173.816,34.904,156.506
C06816=1061.958,327.873,396.968,173.813,34.899,156.505
C06817=1061.951,327.625,397.002,173.809,34.895,156.504
C06818=1061.945,327.377,397.036,173.806,34.890,156.503
C06819=1061.938,327.129,397.070,173.802,34.886,156.502
C06820=1061.932,326.882,397.104,173.798,34.881,156.502
C06821=1061.925,326.634,397.138,173.795,34.876,156.501
C06822=1061.918,326.387,397.172,173.792,34.872,156.500
C06823=1061.912,326.140,397.207,173.788,34.867,156.499
C06824=1061.905,325.892,397.241,173.784,34.863,156.498
C06825=1061.898,325.644,397.275,173.781,34.858,156.497
C06826=1061.892,325.397,397.309,173.777,34.854,156.496
C06827=1061.885,325.149,397.343,173.774,34.850,156.495
C06828=1061.879,324.901,397.377,173.771,34.845,156.494
C06829=1061.873,324.654,397.412,173.766,34.840,156.493
C06830=1061.865,324.406,397.445,173.763,34.836,156.492
C06831=1061.860,324.159,397.479,173.760,34.832,156.491
C06832=1061.852,323.911,397.513,173.757,34.827,156.490
C06833=1061.846,323.663,397.547,173.753,34.822,156.489
C06834=1061.840,323.415,397.581,173.749,34.818,156.488
C06835=1061.833,323.168,397.615,173.746,34.814,156.487
C06836=1061.827,322.921,397.649,173.742,34.809,156.486
C06837=1061.820,322.673,397.683,173.739,34.805,156.485
C06838=1061.814,322.426,397.717,173.736,34.800,156.484
C06839=1061.807,322.178,397.751,173.732,34.796,156.483
C06840=1061.801,321.930,397.784,173.729,34.791,156.483
C06841=1061.795,321.682,397.818,173.725,34.787,156.482
C06842=1061.788,321.435,397.852,173.721,34.782,156.481
C06843=1061.782,321.187,397.886,173.718,34.778,156.480
C06844=1061.775,320.940,397.920,173.715,34.773,156.479
C06845=1061.769,320.691,397.953,173.712,34.769,156.478
C06846=1061.763,320.444,397.987,173.708,34.765,156.477
C06847=1061.756,320.196,398.021,173.705,34.760,156.476
C06848=1061.750,319.949,398.054,173.702,34.756,156.475
C06849=1061.744,319.702,398.088,173.697,34.751,156.474
C06850=1061.737,319.454,398.122,173.694,34.747,156.473
C06851=1061.731,319.206,398.155,173.691,34.742,156.472
C06852=1061.724,318.962,398.189,173.687,34.738,156.472
C06853=1061.718,318.719,398.222,173.684,34.734,156.471
C06854=1061.712,318.475,398.254,173.681,34.729,156.470
C06855=1061.706,318.231,398.288,173.678,34.725,156.469
C06856=1061.700,317.987,398.320,173.674,34.721,156.468
C06857=1061.694,317.744,398.354,173.671,34.717,156.467
C06858=1061.688,317.501,398.387,173.668,34.712,156.466
C06859=1061.681,317.256,398.420,173.664,34.708,156.465
C06860=1061.675,317.009,398.453,173.661,34.703,156.464
C06861=1061.669,316.761,398.487,173.658,34.699,156.463
C06862=1061.662,316.513,398.520,173.655,34.694,156.462
C06863=1061.656,316.266,398.554,173.651,34.690,156.462
C06864=1061.650,316.018,398.586,173.648,34.686,156.461
C06865=1061.643,315.770,398.621,173.645,34.681,156.460
C06866=1061.637,315.522,398.654,173.641,34.677,156.459
C06867=1061.631,315.275,398.688,173.638,34.673,156.458
C06868=1061.625,315.027,398.720,173.635,34.668,156.457
C06869=1061.619,314.780,398.753,173.632,34.664,156.456
C06870=1061.612,314.532,398.788,173.628,34.659,156.455
C06871=1061.606,314.284,398.820,173.625,34.655,156.454
C06872=1061.600,314.036,398.854,173.622,34.650,156.453
C06873=1061.594,313.789,398.887,173.618,34.646,156.452
C06874=1061.587,313.541,398.920,173.614,34.642,156.452
C06875=1061.581,313.294,398.953,173.611,34.638,156.451
C06876=1061.574,313.046,398.986,173.608,34.633,156.450
C06877=1061.567,312.798,399.019,173.604,34.629,156.449
C06878=1061.561,312.550,399.052,173.601,34.625,156.448
C06879=1061.555,312.302,399.084,173.598,34.621,156.447
C06880=1061.548,312.054,399.117,173.595,34.617,156.446
C06881=1061.542,311.807,399.150,173.591,34.613,156.446
C06882=1061.535,311.560,399.184,173.588,34.609,156.445
C06883=1061.529,311.312,399.216,173.585,34.605,156.444
C06884=1061.522,311.064,399.249,173.582,34.600,156.443
C06885=1061.516,310.816,399.282,173.578,34.596,156.442
C06886=1061.509,310.569,399.314,173.575,34.592,156.441
C06887=1061.502,310.321,399.347,173.572,34.587,156.440
C06888=1061.495,310.073,399.380,173.569,34.583,156.439
C06889=1061.489,309.825,399.413,173.565,34.579,156.439
C06890=1061.483,309.577,399.445,173.562,34.575,156.438
C06891=1061.477,309.330,399.478,173.559,34.571,156.437
C06892=1061.470,309.082,399.510,173.556,34.567,156.436
C06893=1061.464,308.834,399.543,173.552,34.563,156.435
C06894=1061.457,308.586,399.576,173.549,34.558,156.434
C06895=1061.450,308.339,399.608,173.546,34.554,156.433
C06896=1061.444,308.091,399.641,173.543,34.550,156.433
C06897=1061.438,307.844,399.674,173.539,34.546,156.432
C06898=1061.432,307.595,399.706,173.536,34.541,156.431
C06899=1061.425,307.348,399.739,173.533,34.537,156.430
C06900=1061.419,307.100,399.771,173.530,34.533,156.429
C06901=1061.413,306.853,399.804,173.527,34.529,156.428
C06902=1061.407,306.605,399.837,173.523,34.525,156.428
C06903=1061.400,306.357,399.868,173.520,34.521,156.427
C06904=1061.393,306.109,399.901,173.517,34.517,156.426
C06905=1061.387,305.861,399.934,173.514,34.513,156.425
C06906=1061.381,305.613,399.966,173.510,34.508,156.424
C06907=1061.374,305.365,399.999,173.508,34.504,156.423
C06908=1061.368,305.124,400.030,173.505,34.500,156.422
C06909=1061.362,304.882,400.062,173.502,34.496,156.422
C06910=1061.356,304.640,400.094,173.498,34.492,156.421
C06911=1061.350,304.399,400.125,173.495,34.488,156.420
C06912=1061.343,304.156,400.157,173.492,34.484,156.419
C06913=1061.337,303.915,400.188,173.489,34.480,156.418
C06914=1061.332,303.673,400.220,173.486,34.476,156.418
C06915=1061.325,303.431,400.252,173.483,34.472,156.417
C06916=1061.318,303.184,400.284,173.480,34.468,156.416
C06917=1061.312,302.935,400.316,173.477,34.464,156.415
C06918=1061.306,302.688,400.349,173.474,34.459,156.414
C06919=1061.301,302.440,400.380,173.470,34.455,156.413
C06920=1061.294,302.193,400.413,173.467,34.451,156.412
C06921=1061.288,301.945,400.445,173.464,34.447,156.412
C06922=1061.281,301.697,400.477,173.461,34.443,156.411
C06923=1061.275,301.449,400.509,173.458,34.439,156.410
C06924=1061.269,301.201,400.542,173.455,34.435,156.409
C06925=1061.262,300.953,400.573,173.452,34.430,156.408
C06926=1061.256,300.705,400.605,173.449,34.426,156.407
C06927=1061.250,300.458,400.638,173.446,34.422,156.407
C06928=1061.245,300.210,400.670,173.442,34.418,156.406
C06929=1061.239,299.962,400.702,173.439,34.414,156.405
C06930=1061.232,299.715,400.734,173.437,34.410,156.404
C06931=1061.226,299.466,400.766,173.434,34.406,156.403
C06932=1061.220,299.218,400.798,173.430,34.401,156.402
C06933=1061.213,298.971,400.831,173.427,34.397,156.402
C06934=1061.207,298.723,400.862,173.424,34.393,156.401
C06935=1061.201,298.475,400.894,173.421,34.389,156.400
C06936=1061.195,298.228,400.927,173.419,34.385,156.399
C06937=1061.188,297.980,400.958,173.415,34.381,156.398
C06938=1061.182,297.731,400.990,173.412,34.376,156.397
C06939=1061.177,297.484,401.022,173.409,34.373,156.397
C06940=1061.171,297.236,401.054,173.406,34.369,156.396
C06941=1061.164,296.988,401.086,173.403,34.365,156.395
C06942=1061.158,296.740,401.118,173.400,34.360,156.394
C06943=1061.151,296.492,401.149,173.397,34.356,156.393
C06944=1061.146,296.245,401.181,173.394,34.352,156.392
C06945=1061.139,295.997,401.213,173.391,34.348,156.392
C06946=1061.133,295.749,401.245,173.388,34.344,156.391
C06947=1061.126,295.501,401.276,173.385,34.340,156.390
C06948=1061.120,295.253,401.308,173.382,34.336,156.389
C06949=1061.114,295.005,401.339,173.379,34.332,156.388
C06950=1061.108,294.757,401.371,173.376,34.328,156.388
C06951=1061.102,294.509,401.403,173.373,34.324,156.387
C06952=1061.095,294.261,401.434,173.369,34.320,156.386
C06953=1061.089,294.014,401.466,173.367,34.316,156.385
C06954=1061.083,293.766,401.497,173.364,34.312,156.384
C06955=1061.076,293.518,401.529,173.361,34.308,156.384
C06956=1061.070,293.270,401.561,173.358,34.304,156.383
C06957=1061.064,293.022,401.591,173.355,34.300,156.382
C06958=1061.057,292.774,401.622,173.352,34.296,156.381
C06959=1061.051,292.526,401.654,173.349,34.292,156.380
C06960=1061.045,292.278,401.686,173.346,34.288,156.380
C06961=1061.039,292.031,401.717,173.343,34.284,156.379
C06962=1061.033,291.783,401.749,173.340,34.280,156.378
C06963=1061.026,291.534,401.780,173.337,34.276,156.377
C06964=1061.020,291.300,401.809,173.334,34.272,156.376
C06965=1061.014,291.066,401.838,173.332,34.269,156.376
C06966=1061.008,290.832,401.868,173.329,34.265,156.375
C06967=1061.002,290.598,401.897,173.325,34.261,156.374
C06968=1060.997,290.363,401.927,173.323,34.257,156.373
C06969=1060.991,290.129,401.957,173.320,34.254,156.373
C06970=1060.985,289.895,401.986,173.318,34.250,156.372
C06971=1060.979,289.661,402.016,173.315,34.246,156.371
C06972=1060.972,289.413,402.047,173.312,34.242,156.370
C06973=1060.966,289.166,402.078,173.309,34.238,156.370
C06974=1060.961,288.917,402.109,173.306,34.234,156.369
C06975=1060.954,288.669,402.141,173.303,34.230,156.368
C06976=1060.948,288.421,402.171,173.300,34.226,156.367
C06977=1060.941,288.173,402.203,173.298,34.222,156.366
C06978=1060.935,287.925,402.233,173.295,34.219,156.366
C06979=1060.929,287.678,402.264,173.291,34.215,156.365
C06980=1060.922,287.429,402.295,173.288,34.211,156.364
C06981=1060.916,287.181,402.327,173.286,34.207,156.363
C06982=1060.910,286.933,402.357,173.283,34.203,156.362
C06983=1060.903,286.685,402.388,173.280,34.199,156.362
C06984=1060.897,286.438,402.419,173.277,34.195,156.361
C06985=1060.890,286.190,402.450,173.274,34.191,156.360
C06986=1060.884,285.941,402.481,173.271,34.187,156.359
C06987=1060.878,285.694,402.512,173.268,34.183,156.359
C06988=1060.872,285.446,402.543,173.266,34.179,156.358
C06989=1060.866,285.197,402.574,173.263,34.176,156.357
C06990=1060.860,284.949,402.605,173.259,34.171,156.356
C06991=1060.854,284.702,402.635,173.257,34.168,156.356
C06992=1060.847,284.453,402.666,173.254,34.164,156.355
C06993=1060.841,284.205,402.698,173.251,34.160,156.354
C06994=1060.835,283.957,402.728,173.249,34.156,156.353
C06995=1060.829,283.709,402.759,173.246,34.152,156.352
C06996=1060.822,283.462,402.790,173.242,34.148,156.352
C06997=1060.816,283.213,402.820,173.240,34.144,156.351
C06998=1060.809,282.966,402.850,173.237,34.140,156.350
C06999=1060.803,282.717,402.881,173.234,34.136,156.349
C07000=1060.797,282.470,402.912,173.232,34.133,156.349
C07001=1060.790,282.221,402.943,173.229,34.128,156.348
C07002=1060.785,281.974,402.973,173.225,34.124,156.347
C07003=1060.779,281.726,403.003,173.223,34.121,156.346
C07004=1060.772,281.477,403.034,173.220,34.116,156.345
C07005=1060.766,281.230,403.065,173.217,34.113,156.345
C07006=1060.760,280.982,403.096,173.215,34.109,156.344
C07007=1060.754,280.734,403.126,173.212,34.105,156.343
C07008=1060.748,280.485,403.157,173.209,34.101,156.342
C07009=1060.742,280.237,403.187,173.206,34.097,156.342
C07010=1060.735,279.989,403.218,173.203,34.093,156.341
C07011=1060.730,279.741,403.248,173.201,34.090,156.340
C07012=1060.724,279.493,403.279,173.198,34.085,156.339
C07013=1060.717,279.245,403.309,173.195,34.082,156.339
C07014=1060.711,278.997,403.339,173.192,34.078,156.338
C07015=1060.704,278.749,403.370,173.189,34.074,156.337
C07016=1060.699,278.501,403.400,173.186,34.070,156.336
C07017=1060.691,278.253,403.430,173.184,34.066,156.335
C07018=1060.686,278.005,403.461,173.181,34.062,156.335
C07019=1060.680,277.757,403.491,173.179,34.058,156.334
C07020=1060.673,277.528,403.519,173.176,34.055,156.333
C07021=1060.668,277.299,403.547,173.173,34.051,156.332
C07022=1060.662,277.070,403.575,173.170,34.047,156.332
C07023=1060.656,276.841,403.603,173.168,34.044,156.331
C07024=1060.651,276.613,403.631,173.166,34.040,156.330
C07025=1060.644,276.384,403.658,173.163,34.037,156.330
C07026=1060.639,276.155,403.686,173.161,34.033,156.329
C07027=1060.634,275.926,403.715,173.158,34.030,156.328
C07028=1060.627,275.678,403.744,173.155,34.026,156.328
C07029=1060.621,275.430,403.775,173.152,34.022,156.327
C07030=1060.615,275.182,403.805,173.150,34.018,156.326
C07031=1060.609,274.934,403.834,173.147,34.014,156.325
C07032=1060.603,274.686,403.865,173.145,34.010,156.324
C07033=1060.596,274.437,403.895,173.142,34.007,156.324
C07034=1060.590,274.189,403.925,173.139,34.003,156.323
C07035=1060.584,273.941,403.955,173.136,33.999,156.322
C07036=1060.577,273.693,403.985,173.133,33.995,156.322
C07037=1060.571,273.445,404.015,173.131,33.991,156.321
C07038=1060.566,273.197,404.045,173.128,33.987,156.320
C07039=1060.559,272.949,404.075,173.126,33.984,156.319
C07040=1060.553,272.701,404.105,173.123,33.980,156.318
C07041=1060.547,272.453,404.134,173.120,33.976,156.318
C07042=1060.541,272.205,404.165,173.117,33.972,156.317
C07043=1060.534,271.956,404.194,173.114,33.968,156.316
C07044=1060.528,271.708,404.225,173.112,33.965,156.316
C07045=1060.522,271.460,404.254,173.109,33.960,156.315
C07046=1060.516,271.212,404.284,173.107,33.957,156.314
C07047=1060.509,270.964,404.314,173.104,33.953,156.313
C07048=1060.503,270.716,404.344,173.102,33.949,156.312
C07049=1060.497,270.468,404.373,173.099,33.945,156.312
C07050=1060.491,270.220,404.403,173.096,33.941,156.311
C07051=1060.484,269.972,404.433,173.093,33.937,156.310
C07052=1060.479,269.723,404.463,173.091,33.934,156.310
C07053=1060.472,269.475,404.492,173.088,33.930,156.309
C07054=1060.467,269.227,404.522,173.086,33.926,156.308
C07055=1060.460,268.978,404.552,173.083,33.922,156.307
C07056=1060.454,268.730,404.582,173.080,33.918,156.306
C07057=1060.448,268.482,404.611,173.077,33.915,156.306
C07058=1060.441,268.234,404.640,173.074,33.911,156.305
C07059=1060.436,267.986,404.670,173.072,33.907,156.304
C07060=1060.429,267.738,404.700,173.069,33.903,156.304
C07061=1060.422,267.489,404.729,173.067,33.900,156.303
C07062=1060.417,267.242,404.759,173.064,33.895,156.302
C07063=1060.410,266.993,404.788,173.062,33.892,156.301
C07064=1060.404,266.745,404.817,173.059,33.888,156.301
C07065=1060.398,266.497,404.848,173.056,33.884,156.300
C07066=1060.391,266.249,404.877,173.053,33.880,156.299
C07067=1060.385,266.001,404.906,173.051,33.877,156.298
C07068=1060.379,265.752,404.935,173.049,33.872,156.298
C07069=1060.373,265.505,404.966,173.046,33.869,156.297
C07070=1060.367,265.256,404.995,173.044,33.865,156.296
C07071=1060.361,265.008,405.024,173.041,33.861,156.295
C07072=1060.355,264.759,405.054,173.039,33.857,156.295
C07073=1060.348,264.511,405.083,173.035,33.854,156.294
C07074=1060.342,264.264,405.112,173.033,33.850,156.293
C07075=1060.335,264.015,405.141,173.030,33.846,156.292
C07076=1060.330,263.788,405.168,173.028,33.842,156.292
C07077=1060.325,263.562,405.195,173.026,33.839,156.291
C07078=1060.319,263.334,405.222,173.023,33.835,156.290
C07079=1060.313,263.108,405.249,173.021,33.832,156.290
C07080=1060.308,262.881,405.275,173.019,33.828,156.289
C07081=1060.301,262.654,405.302,173.017,33.825,156.288
C07082=1060.296,262.427,405.329,173.014,33.822,156.288
C07083=1060.290,262.199,405.355,173.011,33.818,156.287
C07084=1060.284,261.951,405.384,173.009,33.814,156.286
C07085=1060.278,261.703,405.413,173.006,33.811,156.286
C07086=1060.272,261.455,405.442,173.004,33.807,156.285
C07087=1060.265,261.207,405.471,173.001,33.803,156.284
C07088=1060.259,260.959,405.500,172.999,33.799,156.283
C07089=1060.252,260.711,405.529,172.996,33.796,156.283
C07090=1060.245,260.462,405.558,172.994,33.792,156.282
C07091=1060.239,260.214,405.587,172.992,33.788,156.281
C07092=1060.233,259.966,405.616,172.988,33.784,156.280
C07093=1060.226,259.718,405.645,172.986,33.781,156.280
C07094=1060.220,259.469,405.673,172.983,33.777,156.279
C07095=1060.214,259.221,405.702,172.981,33.773,156.278
C07096=1060.208,258.973,405.731,172.978,33.770,156.278
C07097=1060.202,258.724,405.761,172.976,33.765,156.277
C07098=1060.195,258.476,405.790,172.974,33.762,156.276
C07099=1060.189,258.228,405.819,172.971,33.758,156.275
C07100=1060.183,257.979,405.847,172.969,33.755,156.275
C07101=1060.177,257.731,405.876,172.965,33.750,156.274
C07102=1060.171,257.483,405.905,172.963,33.747,156.273
C07103=1060.164,257.235,405.933,172.961,33.743,156.273
C07104=1060.158,256.987,405.962,172.958,33.739,156.272
C07105=1060.152,256.738,405.991,172.956,33.735,156.271
C07106=1060.145,256.490,406.020,172.953,33.732,156.270
C07107=1060.139,256.242,406.048,172.951,33.728,156.270
C07108=1060.133,255.993,406.077,172.949,33.724,156.269
C07109=1060.127,255.745,406.106,172.946,33.720,156.268
C07110=1060.121,255.497,406.135,172.944,33.716,156.267
C07111=1060.115,255.248,406.164,172.940,33.713,156.267
C07112=1060.108,255.001,406.192,172.938,33.709,156.266
C07113=1060.102,254.752,406.220,172.936,33.705,156.265
C07114=1060.096,254.504,406.249,172.933,33.701,156.264
C07115=1060.090,254.255,406.278,172.931,33.698,156.264
C07116=1060.083,254.007,406.307,172.929,33.694,156.263
C07117=1060.077,253.759,406.336,172.926,33.690,156.262
C07118=1060.072,253.511,406.364,172.924,33.686,156.262
C07119=1060.066,253.263,406.393,172.922,33.683,156.261
C07120=1060.059,253.014,406.421,172.919,33.678,156.260
C07121=1060.053,252.766,406.450,172.916,33.675,156.259
C07122=1060.047,252.517,406.478,172.914,33.671,156.259
C07123=1060.040,252.269,406.507,172.911,33.667,156.258
C07124=1060.034,252.020,406.535,172.909,33.663,156.257
C07125=1060.029,251.773,406.564,172.907,33.660,156.256
C07126=1060.022,251.524,406.592,172.904,33.656,156.256
C07127=1060.016,251.276,406.621,172.902,33.652,156.255
C07128=1060.010,251.028,406.649,172.900,33.648,156.254
C07129=1060.004,250.779,406.677,172.897,33.644,156.254
C07130=1059.998,250.531,406.706,172.895,33.640,156.253
C07131=1059.992,250.283,406.734,172.892,33.637,156.252
C07132=1059.985,249.998,406.767,172.889,33.632,156.251
C07133=1059.978,249.713,406.800,172.886,33.627,156.250
C07134=1059.971,249.428,406.832,172.884,33.623,156.249
C07135=1059.964,249.143,406.865,172.881,33.619,156.249
C07136=1059.955,248.801,406.904,172.878,33.614,156.248
C07137=1059.947,248.460,406.943,172.875,33.608,156.247
C07138=1059.941,248.211,406.971,172.872,33.604,156.246
C07139=1059.935,247.962,406.999,172.870,33.601,156.245
C07140=1059.929,247.714,407.028,172.868,33.597,156.244
C07141=1059.924,247.466,407.056,172.865,33.593,156.244
C07142=1059.917,247.217,407.084,172.862,33.589,156.243
C07143=1059.911,246.969,407.112,172.860,33.585,156.242
C07144=1059.905,246.721,407.141,172.858,33.581,156.241
C07145=1059.899,246.473,407.169,172.855,33.577,156.241
C07146=1059.893,246.224,407.197,172.853,33.573,156.240
C07147=1059.887,245.975,407.225,172.851,33.570,156.239
C07148=1059.881,245.727,407.254,172.849,33.566,156.239
C07149=1059.875,245.479,407.281,172.846,33.562,156.238
C07150=1059.869,245.230,407.309,172.844,33.558,156.237
C07151=1059.862,244.982,407.337,172.842,33.555,156.236
C07152=1059.856,244.734,407.366,172.840,33.550,156.235
C07153=1059.850,244.486,407.394,172.836,33.547,156.235
C07154=1059.844,244.237,407.422,172.834,33.543,156.234
C07155=1059.838,243.988,407.450,172.832,33.540,156.233
C07156=1059.832,243.741,407.478,172.829,33.535,156.233
C07157=1059.826,243.492,407.506,172.827,33.532,156.232
C07158=1059.819,243.243,407.534,172.825,33.528,156.231
C07159=1059.814,242.995,407.562,172.823,33.524,156.230
C07160=1059.807,242.747,407.589,172.821,33.520,156.230
C07161=1059.801,242.498,407.618,172.818,33.516,156.229
C07162=1059.795,242.250,407.645,172.816,33.512,156.228
C07163=1059.789,242.002,407.673,172.814,33.509,156.227
C07164=1059.783,241.753,407.701,172.812,33.505,156.227
C07165=1059.776,241.504,407.728,172.809,33.501,156.226
C07166=1059.771,241.256,407.756,172.807,33.497,156.225
C07167=1059.764,241.008,407.784,172.804,33.493,156.225
C07168=1059.757,240.759,407.811,172.802,33.490,156.224
C07169=1059.752,240.511,407.839,172.799,33.486,156.223
C07170=1059.745,240.263,407.867,172.797,33.482,156.222
C07171=1059.739,240.014,407.895,172.795,33.478,156.222
C07172=1059.734,239.766,407.922,172.793,33.475,156.221
C07173=1059.727,239.517,407.950,172.790,33.471,156.220
C07174=1059.721,239.269,407.977,172.788,33.467,156.220
C07175=1059.715,239.021,408.006,172.786,33.463,156.219
C07176=1059.708,238.772,408.033,172.784,33.459,156.218
C07177=1059.703,238.524,408.060,172.782,33.456,156.217
C07178=1059.696,238.275,408.088,172.779,33.451,156.217
C07179=1059.690,238.027,408.116,172.777,33.448,156.216
C07180=1059.684,237.778,408.143,172.775,33.444,156.215
C07181=1059.678,237.530,408.170,172.772,33.440,156.215
C07182=1059.671,237.282,408.198,172.770,33.436,156.214
C07183=1059.665,237.033,408.226,172.767,33.433,156.213
C07184=1059.659,236.784,408.253,172.765,33.429,156.212
C07185=1059.653,236.537,408.280,172.763,33.425,156.212
C07186=1059.648,236.306,408.306,172.761,33.422,156.211
C07187=1059.641,236.074,408.332,172.759,33.418,156.210
C07188=1059.636,235.843,408.357,172.757,33.414,156.210
C07189=1059.630,235.612,408.383,172.755,33.411,156.209
C07190=1059.624,235.381,408.408,172.753,33.407,156.208
C07191=1059.619,235.151,408.433,172.751,33.403,156.207
C07192=1059.613,234.919,408.459,172.749,33.400,156.207
C07193=1059.607,234.688,408.484,172.747,33.397,156.206
C07194=1059.601,234.440,408.512,172.745,33.392,156.205
C07195=1059.595,234.191,408.539,172.742,33.389,156.205
C07196=1059.589,233.943,408.567,172.740,33.385,156.204
C07197=1059.583,233.694,408.594,172.738,33.381,156.203
C07198=1059.577,233.446,408.621,172.735,33.377,156.203
C07199=1059.570,233.197,408.648,172.733,33.373,156.202
C07200=1059.564,232.950,408.675,172.731,33.369,156.201
C07201=1059.559,232.700,408.703,172.729,33.366,156.200
C07202=1059.553,232.452,408.730,172.726,33.362,156.200
C07203=1059.546,232.203,408.757,172.724,33.358,156.199
C07204=1059.541,231.955,408.784,172.722,33.354,156.198
C07205=1059.534,231.707,408.812,172.720,33.350,156.197
C07206=1059.528,231.458,408.838,172.718,33.346,156.197
C07207=1059.521,231.210,408.866,172.716,33.343,156.196
C07208=1059.516,230.961,408.893,172.714,33.339,156.195
C07209=1059.509,230.712,408.920,172.711,33.335,156.194
C07210=1059.503,230.465,408.947,172.709,33.331,156.194
C07211=1059.497,230.216,408.974,172.707,33.327,156.193
C07212=1059.491,229.967,409.001,172.705,33.323,156.192
C07213=1059.485,229.719,409.028,172.703,33.319,156.192
C07214=1059.479,229.470,409.055,172.701,33.316,156.191
C07215=1059.473,229.222,409.082,172.699,33.312,156.190
C07216=1059.466,228.974,409.110,172.697,33.308,156.189
C07217=1059.460,228.725,409.136,172.693,33.304,156.189
C07218=1059.454,228.476,409.163,172.691,33.300,156.188
C07219=1059.448,228.228,409.190,172.689,33.296,156.187
C07220=1059.441,227.979,409.216,172.687,33.293,156.186
C07221=1059.435,227.731,409.244,172.685,33.289,156.186
C07222=1059.429,227.482,409.271,172.683,33.285,156.185
C07223=1059.423,227.234,409.297,172.681,33.281,156.184
C07224=1059.417,226.986,409.324,172.679,33.277,156.184
C07225=1059.411,226.736,409.351,172.677,33.274,156.183
C07226=1059.405,226.489,409.378,172.674,33.269,156.182
C07227=1059.398,226.240,409.405,172.672,33.266,156.181
C07228=1059.392,225.992,409.431,172.670,33.262,156.181
C07229=1059.386,225.743,409.458,172.668,33.258,156.180
C07230=1059.380,225.494,409.485,172.666,33.254,156.179
C07231=1059.374,225.246,409.512,172.664,33.251,156.179
C07232=1059.367,224.998,409.538,172.662,33.246,156.178
C07233=1059.361,224.749,409.565,172.660,33.243,156.177
C07234=1059.355,224.500,409.591,172.658,33.239,156.176
C07235=1059.349,224.252,409.618,172.656,33.235,156.176
C07236=1059.343,224.003,409.645,172.654,33.231,156.175
C07237=1059.337,223.755,409.672,172.652,33.227,156.174
C07238=1059.331,223.507,409.698,172.650,33.223,156.173
C07239=1059.324,223.257,409.725,172.647,33.219,156.173
C07240=1059.319,223.009,409.751,172.645,33.215,156.172
C07241=1059.313,222.761,409.778,172.642,33.212,156.171
C07242=1059.307,222.526,409.804,172.640,33.208,156.170
C07243=1059.300,222.291,409.828,172.638,33.204,156.170
C07244=1059.295,222.056,409.853,172.637,33.201,156.169
C07245=1059.289,221.821,409.879,172.635,33.197,156.168
C07246=1059.283,221.586,409.904,172.633,33.193,156.168
C07247=1059.278,221.351,409.929,172.631,33.190,156.167
C07248=1059.272,221.116,409.955,172.629,33.185,156.166
C07249=1059.266,220.881,409.980,172.627,33.182,156.166
C07250=1059.260,220.633,410.006,172.625,33.178,156.165
C07251=1059.254,220.384,410.032,172.623,33.174,156.164
C07252=1059.247,220.135,410.058,172.621,33.171,156.163
C07253=1059.241,219.887,410.085,172.619,33.166,156.163
C07254=1059.235,219.639,410.111,172.617,33.163,156.162
C07255=1059.229,219.390,410.138,172.615,33.159,156.161
C07256=1059.222,219.141,410.163,172.613,33.155,156.160
C07257=1059.216,218.893,410.190,172.611,33.151,156.160
C07258=1059.211,218.644,410.217,172.609,33.147,156.159
C07259=1059.204,218.396,410.243,172.607,33.143,156.158
C07260=1059.198,218.147,410.270,172.604,33.140,156.158
C07261=1059.191,217.898,410.295,172.602,33.135,156.157
C07262=1059.186,217.650,410.322,172.600,33.132,156.156
C07263=1059.179,217.402,410.348,172.598,33.128,156.155
C07264=1059.173,217.152,410.374,172.596,33.124,156.155
C07265=1059.167,216.904,410.400,172.594,33.120,156.154
C07266=1059.161,216.656,410.427,172.592,33.116,156.153
C07267=1059.155,216.407,410.452,172.590,33.112,156.152
C07268=1059.149,216.159,410.479,172.588,33.108,156.152
C07269=1059.142,215.910,410.505,172.586,33.104,156.151
C07270=1059.136,215.661,410.531,172.584,33.101,156.150
C07271=1059.130,215.413,410.557,172.582,33.096,156.149
C07272=1059.124,215.165,410.584,172.580,33.093,156.149
C07273=1059.118,214.916,410.609,172.578,33.088,156.148
C07274=1059.111,214.667,410.636,172.576,33.085,156.147
C07275=1059.105,214.418,410.661,172.574,33.080,156.146
C07276=1059.099,214.170,410.688,172.573,33.077,156.146
C07277=1059.093,213.921,410.713,172.571,33.073,156.145
C07278=1059.087,213.673,410.740,172.568,33.069,156.144
C07279=1059.081,213.425,410.766,172.566,33.065,156.144
C07280=1059.075,213.176,410.792,172.564,33.061,156.143
